LIN {X 0,Y 254.332,Z 467.701,A -85,B 0,C 180,E1 -18449.998,E2 -18449.998} C_VEL
LIN {X 0,Y 254.199,Z 468.178,A -85,B 0,C 180,E1 -18451.583,E2 -18451.583} C_VEL
LIN {X 0,Y 254.133,Z 468.22,A -85,B 0,C 180,E1 -18453.169,E2 -18453.169} C_VEL
LIN {X 0,Y 254.085,Z 467.695,A -85,B 0,C 180,E1 -18455.277,E2 -18455.277} C_VEL
LIN {X 0,Y 254.253,Z 465.99,A -85,B 0,C 180,E1 -18457.942,E2 -18457.942} C_VEL
LIN {X 0,Y 255.044,Z 462.417,A -85,B 0,C 180,E1 -18461.12,E2 -18461.12} C_VEL
LIN {X 0,Y 256.065,Z 458.576,A -85,B 0,C 180,E1 -18463.489,E2 -18463.489} C_VEL
LIN {X 0,Y 257.677,Z 453.617,A -85,B 0,C 180,E1 -18465.826,E2 -18465.826} C_VEL
LIN {X 0,Y 259.523,Z 447.396,A -85,B 0,C 180,E1 -18468.143,E2 -18468.143} C_VEL
LIN {X 0,Y 261.76,Z 439.641,A -85,B 0,C 180,E1 -18470.427,E2 -18470.427} C_VEL
LIN {X 0,Y 264.683,Z 429.976,A -85,B 0,C 180,E1 -18472.643,E2 -18472.643} C_VEL
LIN {X 0,Y 267.429,Z 419.937,A -85,B 0,C 180,E1 -18474.449,E2 -18474.449} C_VEL
LIN {X 0,Y 270.072,Z 408.613,A -85,B 0,C 180,E1 -18476.047,E2 -18476.047} C_VEL
LIN {X 0,Y 272.396,Z 397.491,A -85,B 0,C 180,E1 -18477.254,E2 -18477.254} C_VEL
LIN {X 0,Y 274.387,Z 386.142,A -85,B 0,C 180,E1 -18478.178,E2 -18478.178} C_VEL
LIN {X 0,Y 276.099,Z 372.699,A -85,B 0,C 180,E1 -18478.953,E2 -18478.953} C_VEL
LIN {X 0,Y 277.011,Z 360.119,A -85,B 0,C 180,E1 -18479.424,E2 -18479.424} C_VEL
LIN {X 0,Y 278.882,Z 309.876,A -85,B 0,C 180,E1 -18480.736,E2 -18480.736} C_VEL
LIN {X 0,Y 275.996,Z 287.607,A -85,B 0,C 180,E1 -18481.882,E2 -18481.882} C_VEL
LIN {X 0,Y 273.894,Z 274.147,A -85,B 0,C 180,E1 -18482.654,E2 -18482.654} C_VEL
LIN {X 0,Y 266.764,Z 255.183,A -85,B 0,C 180,E1 -18484.501,E2 -18484.501} C_VEL
LIN {X 0,Y 260.562,Z 245.546,A -85,B 0,C 180,E1 -18485.985,E2 -18485.985} C_VEL
LIN {X 0,Y 258.11,Z 241.688,A -85,B 0,C 180,E1 -18486.642,E2 -18486.642} C_VEL
LIN {X 0,Y 256.399,Z 238.938,A -85,B 0,C 180,E1 -18487.143,E2 -18487.143} C_VEL
LIN {X 0,Y 256.108,Z 237.583,A -85,B 0,C 180,E1 -18487.317,E2 -18487.317} C_VEL
LIN {X 0,Y 256.024,Z 237.584,A -85,B 0,C 180,E1 -18492.17,E2 -18492.17} C_VEL
LIN {X 0,Y 256.015,Z 237.588,A -85,B 0,C 180,E1 -18496.663,E2 -18496.663} C_VEL
LIN {X 0,Y 256.059,Z 237.588,A -85,B 0,C 180,E1 -18500.856,E2 -18500.856} C_VEL
LIN {X 0,Y 256.118,Z 237.562,A -85,B 0,C 180,E1 -18502.866,E2 -18502.866} C_VEL
LIN {X 0,Y 256.058,Z 237.583,A -85,B 0,C 180,E1 -18506.706,E2 -18506.706} C_VEL
LIN {X 0,Y 256.032,Z 237.558,A -85,B 0,C 180,E1 -18510.39,E2 -18510.39} C_VEL
LIN {X 0,Y 256.122,Z 237.573,A -85,B 0,C 180,E1 -18514.889,E2 -18514.889} C_VEL
LIN {X 0,Y 256.115,Z 237.547,A -85,B 0,C 180,E1 -18519.101,E2 -18519.101} C_VEL
LIN {X 0,Y 256.222,Z 237.547,A -85,B 0,C 180,E1 -18524.08,E2 -18524.08} C_VEL
LIN {X 0,Y 256.282,Z 237.553,A -85,B 0,C 180,E1 -18528.933,E2 -18528.933} C_VEL
LIN {X 0,Y 256.459,Z 237.526,A -85,B 0,C 180,E1 -18532.125,E2 -18532.125} C_VEL
LIN {X 0,Y 256.451,Z 237.522,A -85,B 0,C 180,E1 -18536.858,E2 -18536.858} C_VEL
LIN {X 0,Y 256.691,Z 237.508,A -85,B 0,C 180,E1 -18538.431,E2 -18538.431} C_VEL
LIN {X 0,Y 256.694,Z 237.476,A -85,B 0,C 180,E1 -18541.569,E2 -18541.569} C_VEL
LIN {X 0,Y 256.461,Z 237.529,A -85,B 0,C 180,E1 -18546.735,E2 -18546.735} C_VEL
LIN {X 0,Y 256.419,Z 237.512,A -85,B 0,C 180,E1 -18549.466,E2 -18549.466} C_VEL
LIN {X 0,Y 256.231,Z 237.564,A -85,B 0,C 180,E1 -18554.292,E2 -18554.292} C_VEL
LIN {X 0,Y 256.175,Z 237.545,A -85,B 0,C 180,E1 -18557.565,E2 -18557.565} C_VEL
LIN {X 0,Y 256.15,Z 237.578,A -85,B 0,C 180,E1 -18561.121,E2 -18561.121} C_VEL
LIN {X 0,Y 256.182,Z 237.56,A -85,B 0,C 180,E1 -18565.14,E2 -18565.14} C_VEL
LIN {X 0,Y 256.098,Z 237.567,A -85,B 0,C 180,E1 -18569.602,E2 -18569.602} C_VEL
LIN {X 0,Y 256.062,Z 237.579,A -85,B 0,C 180,E1 -18573.294,E2 -18573.294} C_VEL
LIN {X 0,Y 256.116,Z 237.579,A -85,B 0,C 180,E1 -18577.274,E2 -18577.274} C_VEL
LIN {X 0,Y 256.071,Z 237.583,A -85,B 0,C 180,E1 -18579.238,E2 -18579.238} C_VEL
LIN {X 0,Y 257.093,Z 240.49,A -85,B 0,C 180,E1 -18579.558,E2 -18579.558} C_VEL
LIN {X 0,Y 259.057,Z 242.91,A -85,B 0,C 180,E1 -18580.037,E2 -18580.037} C_VEL
LIN {X 0,Y 261.326,Z 246.338,A -85,B 0,C 180,E1 -18580.6,E2 -18580.6} C_VEL
LIN {X 0,Y 270.947,Z 261.865,A -85,B 0,C 180,E1 -18582.863,E2 -18582.863} C_VEL
LIN {X 0,Y 279.224,Z 277.008,A -85,B 0,C 180,E1 -18584.684,E2 -18584.684} C_VEL
LIN {X 0,Y 280.664,Z 279.841,A -85,B 0,C 180,E1 -18584.991,E2 -18584.991} C_VEL
LIN {X 0,Y 277.97,Z 342.078,A -85,B 0,C 180,E1 -18586.575,E2 -18586.575} C_VEL
LIN {X 0,Y 276.996,Z 355.523,A -85,B 0,C 180,E1 -18587.178,E2 -18587.178} C_VEL
LIN {X 0,Y 275.637,Z 367.061,A -85,B 0,C 180,E1 -18587.947,E2 -18587.947} C_VEL
LIN {X 0,Y 273.694,Z 379.563,A -85,B 0,C 180,E1 -18589.098,E2 -18589.098} C_VEL
LIN {X 0,Y 271.536,Z 390.525,A -85,B 0,C 180,E1 -18590.408,E2 -18590.408} C_VEL
LIN {X 0,Y 268.892,Z 401.605,A -85,B 0,C 180,E1 -18592.107,E2 -18592.107} C_VEL
LIN {X 0,Y 266.236,Z 411.466,A -85,B 0,C 180,E1 -18594.033,E2 -18594.033} C_VEL
LIN {X 0,Y 263.862,Z 419.47,A -85,B 0,C 180,E1 -18595.992,E2 -18595.992} C_VEL
LIN {X 0,Y 261.372,Z 427.169,A -85,B 0,C 180,E1 -18598.379,E2 -18598.379} C_VEL
LIN {X 0,Y 259.283,Z 433.28,A -85,B 0,C 180,E1 -18600.8,E2 -18600.8} C_VEL
LIN {X 0,Y 257.608,Z 438.031,A -85,B 0,C 180,E1 -18603.249,E2 -18603.249} C_VEL
LIN {X 0,Y 256.26,Z 441.573,A -85,B 0,C 180,E1 -18605.711,E2 -18605.711} C_VEL
LIN {X 0,Y 255.556,Z 443.304,A -85,B 0,C 180,E1 -18607.358,E2 -18607.358} C_VEL
LIN {X 0,Y 254.774,Z 445.019,A -85,B 0,C 180,E1 -18609.703,E2 -18609.703} C_VEL
LIN {X 0,Y 254.185,Z 445.88,A -85,B 0,C 180,E1 -18612.295,E2 -18612.295} C_VEL
LIN {X 0,Y 254.019,Z 445.872,A -85,B 0,C 180,E1 -18613.94,E2 -18613.94} C_VEL
LIN {X 0,Y 253.95,Z 445.458,A -85,B 0,C 180,E1 -18615.61,E2 -18615.61} C_VEL
LIN {X 0,Y 253.929,Z 444.63,A -85,B 0,C 180,E1 -18617.21,E2 -18617.21} C_VEL
LIN {X 0,Y 253.971,Z 443.362,A -85,B 0,C 180,E1 -18618.833,E2 -18618.833} C_VEL
LIN {X 0,Y 254.283,Z 440.661,A -85,B 0,C 180,E1 -18621.258,E2 -18621.258} C_VEL
LIN {X 0,Y 254.758,Z 436.93,A -85,B 0,C 180,E1 -18623.666,E2 -18623.666} C_VEL
LIN {X 0,Y 255.357,Z 432.082,A -85,B 0,C 180,E1 -18626.056,E2 -18626.056} C_VEL
LIN {X 0,Y 256.233,Z 425.967,A -85,B 0,C 180,E1 -18628.43,E2 -18628.43} C_VEL
LIN {X 0,Y 257.432,Z 418.31,A -85,B 0,C 180,E1 -18630.784,E2 -18630.784} C_VEL
LIN {X 0,Y 258.949,Z 408.727,A -85,B 0,C 180,E1 -18633.113,E2 -18633.113} C_VEL
LIN {X 0,Y 260.486,Z 398.784,A -85,B 0,C 180,E1 -18635.032,E2 -18635.032} C_VEL
LIN {X 0,Y 262.061,Z 387.521,A -85,B 0,C 180,E1 -18636.749,E2 -18636.749} C_VEL
LIN {X 0,Y 263.373,Z 376.65,A -85,B 0,C 180,E1 -18638.055,E2 -18638.055} C_VEL
LIN {X 0,Y 264.412,Z 364.482,A -85,B 0,C 180,E1 -18639.178,E2 -18639.178} C_VEL
LIN {X 0,Y 265.375,Z 350.98,A -85,B 0,C 180,E1 -18640.058,E2 -18640.058} C_VEL
LIN {X 0,Y 265.953,Z 338.628,A -85,B 0,C 180,E1 -18640.565,E2 -18640.565} C_VEL
LIN {X 0,Y 268.031,Z 266.062,A -85,B 0,C 180,E1 -18642.468,E2 -18642.468} C_VEL
LIN {X 0,Y 258.649,Z 243.319,A -85,B 0,C 180,E1 -18643.978,E2 -18643.978} C_VEL
LIN {X 0,Y 256.398,Z 238.283,A -85,B 0,C 180,E1 -18644.346,E2 -18644.346} C_VEL
LIN {X 0,Y 256.287,Z 237.561,A -85,B 0,C 180,E1 -18644.391,E2 -18644.391} C_VEL
LIN {X 0,Y 256.216,Z 237.569,A -85,B 0,C 180,E1 -18647.563,E2 -18647.563} C_VEL
LIN {X 0,Y 256.157,Z 237.576,A -85,B 0,C 180,E1 -18651.117,E2 -18651.117} C_VEL
LIN {X 0,Y 256.092,Z 237.584,A -85,B 0,C 180,E1 -18655.091,E2 -18655.091} C_VEL
LIN {X 0,Y 256.082,Z 237.586,A -85,B 0,C 180,E1 -18658.57,E2 -18658.57} C_VEL
LIN {X 0,Y 256.076,Z 237.584,A -85,B 0,C 180,E1 -18661.701,E2 -18661.701} C_VEL
LIN {X 0,Y 256.085,Z 237.584,A -85,B 0,C 180,E1 -18665.194,E2 -18665.194} C_VEL
LIN {X 0,Y 256.111,Z 237.578,A -85,B 0,C 180,E1 -18667.268,E2 -18667.268} C_VEL
LIN {X 0,Y 256.025,Z 237.592,A -85,B 0,C 180,E1 -18671.211,E2 -18671.211} C_VEL
LIN {X 0,Y 256.024,Z 237.593,A -85,B 0,C 180,E1 -18675.54,E2 -18675.54} C_VEL
LIN {X 0,Y 256.015,Z 237.592,A -85,B 0,C 180,E1 -18678.788,E2 -18678.788} C_VEL
LIN {X 0,Y 256.105,Z 237.573,A -85,B 0,C 180,E1 -18682.862,E2 -18682.862} C_VEL
LIN {X 0,Y 256.072,Z 237.586,A -85,B 0,C 180,E1 -18686.707,E2 -18686.707} C_VEL
LIN {X 0,Y 256.048,Z 237.582,A -85,B 0,C 180,E1 -18690.391,E2 -18690.391} C_VEL
LIN {X 0,Y 256.189,Z 237.561,A -85,B 0,C 180,E1 -18694.127,E2 -18694.127} C_VEL
LIN {X 0,Y 263.357,Z 264.994,A -85,B 0,C 180,E1 -18695.646,E2 -18695.646} C_VEL
LIN {X 0,Y 260.067,Z 344.326,A -85,B 0,C 180,E1 -18699.122,E2 -18699.122} C_VEL
LIN {X 0,Y 259.667,Z 354.656,A -85,B 0,C 180,E1 -18699.772,E2 -18699.772} C_VEL
LIN {X 0,Y 259.079,Z 358.355,A -85,B 0,C 180,E1 -18700.042,E2 -18700.042} C_VEL
LIN {X 0,Y 256.709,Z 365.442,A -85,B 0,C 180,E1 -18700.625,E2 -18700.625} C_VEL
LIN {X 0,Y 251.786,Z 377.309,A -85,B 0,C 180,E1 -18701.837,E2 -18701.837} C_VEL
LIN {X 0,Y 250.816,Z 382.417,A -85,B 0,C 180,E1 -18702.475,E2 -18702.475} C_VEL
LIN {X 0,Y 249.822,Z 394.701,A -85,B 0,C 180,E1 -18704.289,E2 -18704.289} C_VEL
LIN {X 0,Y 249.018,Z 405.731,A -85,B 0,C 180,E1 -18706.327,E2 -18706.327} C_VEL
LIN {X 0,Y 248.245,Z 415.577,A -85,B 0,C 180,E1 -18708.569,E2 -18708.569} C_VEL
LIN {X 0,Y 247.677,Z 424.27,A -85,B 0,C 180,E1 -18711.021,E2 -18711.021} C_VEL
LIN {X 0,Y 247.325,Z 431.278,A -85,B 0,C 180,E1 -18713.473,E2 -18713.473} C_VEL
LIN {X 0,Y 247.134,Z 436.857,A -85,B 0,C 180,E1 -18715.923,E2 -18715.923} C_VEL
LIN {X 0,Y 247.098,Z 441.202,A -85,B 0,C 180,E1 -18718.37,E2 -18718.37} C_VEL
LIN {X 0,Y 247.115,Z 443.466,A -85,B 0,C 180,E1 -18720,E2 -18720} C_VEL
LIN {X 0,Y 247.28,Z 445.312,A -85,B 0,C 180,E1 -18721.628,E2 -18721.628} C_VEL
LIN {X 0,Y 247.577,Z 446.731,A -85,B 0,C 180,E1 -18723.254,E2 -18723.254} C_VEL
LIN {X 0,Y 248.038,Z 447.698,A -85,B 0,C 180,E1 -18724.876,E2 -18724.876} C_VEL
LIN {X 0,Y 248.591,Z 448.265,A -85,B 0,C 180,E1 -18726.493,E2 -18726.493} C_VEL
LIN {X 0,Y 249.827,Z 448.254,A -85,B 0,C 180,E1 -18729.717,E2 -18729.717} C_VEL
LIN {X 0,Y 251.109,Z 447.597,A -85,B 0,C 180,E1 -18731.298,E2 -18731.298} C_VEL
LIN {X 0,Y 253.831,Z 445.101,A -85,B 0,C 180,E1 -18734.429,E2 -18734.429} C_VEL
LIN {X 0,Y 256.335,Z 442.134,A -85,B 0,C 180,E1 -18736.731,E2 -18736.731} C_VEL
LIN {X 0,Y 259.287,Z 438.171,A -85,B 0,C 180,E1 -18738.981,E2 -18738.981} C_VEL
LIN {X 0,Y 262.632,Z 433.126,A -85,B 0,C 180,E1 -18741.177,E2 -18741.177} C_VEL
LIN {X 0,Y 267.091,Z 425.702,A -85,B 0,C 180,E1 -18743.658,E2 -18743.658} C_VEL
LIN {X 0,Y 271.348,Z 417.742,A -85,B 0,C 180,E1 -18745.711,E2 -18745.711} C_VEL
LIN {X 0,Y 276.046,Z 408.045,A -85,B 0,C 180,E1 -18747.687,E2 -18747.687} C_VEL
LIN {X 0,Y 281.008,Z 396.101,A -85,B 0,C 180,E1 -18749.6,E2 -18749.6} C_VEL
LIN {X 0,Y 285.073,Z 384.991,A -85,B 0,C 180,E1 -18750.973,E2 -18750.973} C_VEL
LIN {X 0,Y 289.312,Z 371.238,A -85,B 0,C 180,E1 -18752.305,E2 -18752.305} C_VEL
LIN {X 0,Y 292.512,Z 358.436,A -85,B 0,C 180,E1 -18753.237,E2 -18753.237} C_VEL
LIN {X 0,Y 295.48,Z 343.206,A -85,B 0,C 180,E1 -18754.034,E2 -18754.034} C_VEL
LIN {X 0,Y 301.355,Z 311.174,A -85,B 0,C 180,E1 -18755.455,E2 -18755.455} C_VEL
LIN {X 0,Y 299.414,Z 306.995,A -85,B 0,C 180,E1 -18757.257,E2 -18757.257} C_VEL
LIN {X 0,Y 297.784,Z 304.069,A -85,B 0,C 180,E1 -18759.174,E2 -18759.174} C_VEL
LIN {X 0,Y 296.428,Z 302.2,A -85,B 0,C 180,E1 -18761.594,E2 -18761.594} C_VEL
LIN {X 0,Y 295.823,Z 302.186,A -85,B 0,C 180,E1 -18764.141,E2 -18764.141} C_VEL
LIN {X 0,Y 296.142,Z 303.62,A -85,B 0,C 180,E1 -18766.508,E2 -18766.508} C_VEL
LIN {X 0,Y 297.699,Z 309.061,A -85,B 0,C 180,E1 -18769.834,E2 -18769.834} C_VEL
LIN {X 0,Y 299.099,Z 314.072,A -85,B 0,C 180,E1 -18771.679,E2 -18771.679} C_VEL
LIN {X 0,Y 300.196,Z 318.243,A -85,B 0,C 180,E1 -18772.887,E2 -18772.887} C_VEL
LIN {X 0,Y 299.894,Z 322.243,A -85,B 0,C 180,E1 -18773.274,E2 -18773.274} C_VEL
LIN {X 0,Y 292.23,Z 364.761,A -85,B 0,C 180,E1 -18775.205,E2 -18775.205} C_VEL
LIN {X 0,Y 288.932,Z 378.053,A -85,B 0,C 180,E1 -18775.98,E2 -18775.98} C_VEL
LIN {X 0,Y 284.499,Z 392.348,A -85,B 0,C 180,E1 -18777.078,E2 -18777.078} C_VEL
LIN {X 0,Y 279.95,Z 404.975,A -85,B 0,C 180,E1 -18778.394,E2 -18778.394} C_VEL
LIN {X 0,Y 275.251,Z 416.507,A -85,B 0,C 180,E1 -18779.926,E2 -18779.926} C_VEL
LIN {X 0,Y 270.494,Z 426.944,A -85,B 0,C 180,E1 -18781.693,E2 -18781.693} C_VEL
LIN {X 0,Y 265.894,Z 436.393,A -85,B 0,C 180,E1 -18783.72,E2 -18783.72} C_VEL
LIN {X 0,Y 261.761,Z 444.205,A -85,B 0,C 180,E1 -18785.828,E2 -18785.828} C_VEL
LIN {X 0,Y 257.839,Z 451.045,A -85,B 0,C 180,E1 -18788.148,E2 -18788.148} C_VEL
LIN {X 0,Y 254.56,Z 456.733,A -85,B 0,C 180,E1 -18790.651,E2 -18790.651} C_VEL
LIN {X 0,Y 252.133,Z 460.809,A -85,B 0,C 180,E1 -18792.98,E2 -18792.98} C_VEL
LIN {X 0,Y 250.014,Z 463.933,A -85,B 0,C 180,E1 -18795.343,E2 -18795.343} C_VEL
LIN {X 0,Y 248.239,Z 466.66,A -85,B 0,C 180,E1 -18798.568,E2 -18798.568} C_VEL
LIN {X 0,Y 247.649,Z 467.451,A -85,B 0,C 180,E1 -18800.195,E2 -18800.195} C_VEL
LIN {X 0,Y 247.249,Z 467.829,A -85,B 0,C 180,E1 -18801.827,E2 -18801.827} C_VEL
LIN {X 0,Y 247.039,Z 467.373,A -85,B 0,C 180,E1 -18805.102,E2 -18805.102} C_VEL
LIN {X 0,Y 247.16,Z 465.954,A -85,B 0,C 180,E1 -18807.757,E2 -18807.757} C_VEL
LIN {X 0,Y 247.247,Z 467.319,A -85,B 0,C 180,E1 -18809.998,E2 -18809.998} C_VEL
LIN {X 0,Y 247.121,Z 467.839,A -85,B 0,C 180,E1 -18811.628,E2 -18811.628} C_VEL
LIN {X 0,Y 247.042,Z 467.918,A -85,B 0,C 180,E1 -18813.26,E2 -18813.26} C_VEL
LIN {X 0,Y 246.989,Z 467.503,A -85,B 0,C 180,E1 -18815.18,E2 -18815.18} C_VEL
LIN {X 0,Y 247.192,Z 465.788,A -85,B 0,C 180,E1 -18818.171,E2 -18818.171} C_VEL
LIN {X 0,Y 247.562,Z 464.242,A -85,B 0,C 180,E1 -18819.805,E2 -18819.805} C_VEL
LIN {X 0,Y 248.34,Z 461.149,A -85,B 0,C 180,E1 -18822.252,E2 -18822.252} C_VEL
LIN {X 0,Y 249.652,Z 457.016,A -85,B 0,C 180,E1 -18824.675,E2 -18824.675} C_VEL
LIN {X 0,Y 251.72,Z 450.712,A -85,B 0,C 180,E1 -18827.464,E2 -18827.464} C_VEL
LIN {X 0,Y 253.809,Z 443.996,A -85,B 0,C 180,E1 -18829.784,E2 -18829.784} C_VEL
LIN {X 0,Y 256.089,Z 436.905,A -85,B 0,C 180,E1 -18831.744,E2 -18831.744} C_VEL
LIN {X 0,Y 258.737,Z 428.501,A -85,B 0,C 180,E1 -18833.617,E2 -18833.617} C_VEL
LIN {X 0,Y 261.625,Z 418.133,A -85,B 0,C 180,E1 -18835.453,E2 -18835.453} C_VEL
LIN {X 0,Y 264.379,Z 406.492,A -85,B 0,C 180,E1 -18837.078,E2 -18837.078} C_VEL
LIN {X 0,Y 266.878,Z 394.749,A -85,B 0,C 180,E1 -18838.293,E2 -18838.293} C_VEL
LIN {X 0,Y 268.992,Z 382.582,A -85,B 0,C 180,E1 -18839.224,E2 -18839.224} C_VEL
LIN {X 0,Y 270.49,Z 370.041,A -85,B 0,C 180,E1 -18839.907,E2 -18839.907} C_VEL
LIN {X 0,Y 271.362,Z 355.831,A -85,B 0,C 180,E1 -18840.383,E2 -18840.383} C_VEL
LIN {X 0,Y 273.145,Z 310.97,A -85,B 0,C 180,E1 -18841.566,E2 -18841.566} C_VEL
LIN {X 0,Y 269.842,Z 284.972,A -85,B 0,C 180,E1 -18842.957,E2 -18842.957} C_VEL
LIN {X 0,Y 268.523,Z 276.891,A -85,B 0,C 180,E1 -18843.451,E2 -18843.451} C_VEL
LIN {X 0,Y 262.058,Z 259.465,A -85,B 0,C 180,E1 -18845.202,E2 -18845.202} C_VEL
LIN {X 0,Y 255.922,Z 249.902,A -85,B 0,C 180,E1 -18846.737,E2 -18846.737} C_VEL
LIN {X 0,Y 253.701,Z 246.502,A -85,B 0,C 180,E1 -18847.321,E2 -18847.321} C_VEL
LIN {X 0,Y 251.394,Z 242.907,A -85,B 0,C 180,E1 -18847.952,E2 -18847.952} C_VEL
LIN {X 0,Y 249.561,Z 240.46,A -85,B 0,C 180,E1 -18848.494,E2 -18848.494} C_VEL
LIN {X 0,Y 249.019,Z 238.452,A -85,B 0,C 180,E1 -18848.781,E2 -18848.781} C_VEL
LIN {X 0,Y 248.961,Z 238.458,A -85,B 0,C 180,E1 -18852.781,E2 -18852.781} C_VEL
LIN {X 0,Y 248.972,Z 238.455,A -85,B 0,C 180,E1 -18857.354,E2 -18857.354} C_VEL
LIN {X 0,Y 249.032,Z 238.454,A -85,B 0,C 180,E1 -18862.2,E2 -18862.2} C_VEL
LIN {X 0,Y 249.035,Z 238.445,A -85,B 0,C 180,E1 -18865.638,E2 -18865.638} C_VEL
LIN {X 0,Y 248.985,Z 238.442,A -85,B 0,C 180,E1 -18869.464,E2 -18869.464} C_VEL
LIN {X 0,Y 249.015,Z 238.453,A -85,B 0,C 180,E1 -18873.156,E2 -18873.156} C_VEL
LIN {X 0,Y 249.043,Z 238.43,A -85,B 0,C 180,E1 -18876.729,E2 -18876.729} C_VEL
LIN {X 0,Y 249.05,Z 238.443,A -85,B 0,C 180,E1 -18880.207,E2 -18880.207} C_VEL
LIN {X 0,Y 249.168,Z 238.433,A -85,B 0,C 180,E1 -18883.617,E2 -18883.617} C_VEL
LIN {X 0,Y 249.225,Z 238.428,A -85,B 0,C 180,E1 -18888.616,E2 -18888.616} C_VEL
LIN {X 0,Y 249.408,Z 238.406,A -85,B 0,C 180,E1 -18891.901,E2 -18891.901} C_VEL
LIN {X 0,Y 249.258,Z 238.397,A -85,B 0,C 180,E1 -18895.148,E2 -18895.148} C_VEL
LIN {X 0,Y 249.652,Z 238.384,A -85,B 0,C 180,E1 -18898.387,E2 -18898.387} C_VEL
LIN {X 0,Y 249.654,Z 238.352,A -85,B 0,C 180,E1 -18901.614,E2 -18901.614} C_VEL
LIN {X 0,Y 249.43,Z 238.406,A -85,B 0,C 180,E1 -18906.72,E2 -18906.72} C_VEL
LIN {X 0,Y 249.335,Z 238.391,A -85,B 0,C 180,E1 -18909.737,E2 -18909.737} C_VEL
LIN {X 0,Y 249.176,Z 238.441,A -85,B 0,C 180,E1 -18914.706,E2 -18914.706} C_VEL
LIN {X 0,Y 249.112,Z 238.427,A -85,B 0,C 180,E1 -18918.08,E2 -18918.08} C_VEL
LIN {X 0,Y 249.08,Z 238.454,A -85,B 0,C 180,E1 -18921.519,E2 -18921.519} C_VEL
LIN {X 0,Y 249.125,Z 238.444,A -85,B 0,C 180,E1 -18925.483,E2 -18925.483} C_VEL
LIN {X 0,Y 249.067,Z 238.442,A -85,B 0,C 180,E1 -18928.99,E2 -18928.99} C_VEL
LIN {X 0,Y 249.025,Z 238.465,A -85,B 0,C 180,E1 -18932.427,E2 -18932.427} C_VEL
LIN {X 0,Y 249.103,Z 238.454,A -85,B 0,C 180,E1 -18937.107,E2 -18937.107} C_VEL
LIN {X 0,Y 249.057,Z 238.556,A -85,B 0,C 180,E1 -18937.784,E2 -18937.784} C_VEL
LIN {X 0,Y 249.971,Z 241.201,A -85,B 0,C 180,E1 -18938.091,E2 -18938.091} C_VEL
LIN {X 0,Y 252.166,Z 243.937,A -85,B 0,C 180,E1 -18938.671,E2 -18938.671} C_VEL
LIN {X 0,Y 254.332,Z 247.247,A -85,B 0,C 180,E1 -18939.251,E2 -18939.251} C_VEL
LIN {X 0,Y 262.484,Z 259.993,A -85,B 0,C 180,E1 -18941.306,E2 -18941.306} C_VEL
LIN {X 0,Y 269.485,Z 271.94,A -85,B 0,C 180,E1 -18942.955,E2 -18942.955} C_VEL
LIN {X 0,Y 274.859,Z 282.268,A -85,B 0,C 180,E1 -18944.174,E2 -18944.174} C_VEL
LIN {X 0,Y 272.142,Z 342.694,A -85,B 0,C 180,E1 -18945.741,E2 -18945.741} C_VEL
LIN {X 0,Y 271.116,Z 356.115,A -85,B 0,C 180,E1 -18946.359,E2 -18946.359} C_VEL
LIN {X 0,Y 269.686,Z 367.66,A -85,B 0,C 180,E1 -18947.149,E2 -18947.149} C_VEL
LIN {X 0,Y 267.779,Z 379.415,A -85,B 0,C 180,E1 -18948.245,E2 -18948.245} C_VEL
LIN {X 0,Y 265.531,Z 390.455,A -85,B 0,C 180,E1 -18949.577,E2 -18949.577} C_VEL
LIN {X 0,Y 262.939,Z 401.008,A -85,B 0,C 180,E1 -18951.196,E2 -18951.196} C_VEL
LIN {X 0,Y 260.246,Z 410.628,A -85,B 0,C 180,E1 -18953.07,E2 -18953.07} C_VEL
LIN {X 0,Y 257.703,Z 418.826,A -85,B 0,C 180,E1 -18955.063,E2 -18955.063} C_VEL
LIN {X 0,Y 255.483,Z 425.56,A -85,B 0,C 180,E1 -18957.094,E2 -18957.094} C_VEL
LIN {X 0,Y 253.352,Z 431.504,A -85,B 0,C 180,E1 -18959.311,E2 -18959.311} C_VEL
LIN {X 0,Y 251.523,Z 436.428,A -85,B 0,C 180,E1 -18961.642,E2 -18961.642} C_VEL
LIN {X 0,Y 249.986,Z 440.404,A -85,B 0,C 180,E1 -18964.112,E2 -18964.112} C_VEL
LIN {X 0,Y 248.724,Z 443.392,A -85,B 0,C 180,E1 -18966.7,E2 -18966.7} C_VEL
LIN {X 0,Y 247.754,Z 445.352,A -85,B 0,C 180,E1 -18969.41,E2 -18969.41} C_VEL
LIN {X 0,Y 247.174,Z 446.175,A -85,B 0,C 180,E1 -18971.776,E2 -18971.776} C_VEL
LIN {X 0,Y 246.977,Z 446.22,A -85,B 0,C 180,E1 -18973.469,E2 -18973.469} C_VEL
LIN {X 0,Y 246.87,Z 445.775,A -85,B 0,C 180,E1 -18975.452,E2 -18975.452} C_VEL
LIN {X 0,Y 246.857,Z 443.911,A -85,B 0,C 180,E1 -18978.506,E2 -18978.506} C_VEL
LIN {X 0,Y 247.143,Z 441.315,A -85,B 0,C 180,E1 -18981.004,E2 -18981.004} C_VEL
LIN {X 0,Y 247.623,Z 437.693,A -85,B 0,C 180,E1 -18983.483,E2 -18983.483} C_VEL
LIN {X 0,Y 248.211,Z 432.963,A -85,B 0,C 180,E1 -18985.943,E2 -18985.943} C_VEL
LIN {X 0,Y 249.095,Z 426.976,A -85,B 0,C 180,E1 -18988.385,E2 -18988.385} C_VEL
LIN {X 0,Y 250.328,Z 419.518,A -85,B 0,C 180,E1 -18990.806,E2 -18990.806} C_VEL
LIN {X 0,Y 251.559,Z 411.884,A -85,B 0,C 180,E1 -18992.804,E2 -18992.804} C_VEL
LIN {X 0,Y 253.216,Z 401.518,A -85,B 0,C 180,E1 -18994.977,E2 -18994.977} C_VEL
LIN {X 0,Y 254.889,Z 390.698,A -85,B 0,C 180,E1 -18996.775,E2 -18996.775} C_VEL
LIN {X 0,Y 256.372,Z 379.085,A -85,B 0,C 180,E1 -18998.276,E2 -18998.276} C_VEL
LIN {X 0,Y 257.517,Z 366.588,A -85,B 0,C 180,E1 -18999.525,E2 -18999.525} C_VEL
LIN {X 0,Y 258.56,Z 353.781,A -85,B 0,C 180,E1 -19000.425,E2 -19000.425} C_VEL
LIN {X 0,Y 259.228,Z 340.348,A -85,B 0,C 180,E1 -19001.041,E2 -19001.041} C_VEL
LIN {X 0,Y 261.373,Z 267.559,A -85,B 0,C 180,E1 -19003.007,E2 -19003.007} C_VEL
LIN {X 0,Y 252.476,Z 246.187,A -85,B 0,C 180,E1 -19004.489,E2 -19004.489} C_VEL
LIN {X 0,Y 249.472,Z 239.544,A -85,B 0,C 180,E1 -19004.997,E2 -19004.997} C_VEL
LIN {X 0,Y 249.251,Z 238.437,A -85,B 0,C 180,E1 -19005.068,E2 -19005.068} C_VEL
LIN {X 0,Y 249.145,Z 238.45,A -85,B 0,C 180,E1 -19008.079,E2 -19008.079} C_VEL
LIN {X 0,Y 249.088,Z 238.457,A -85,B 0,C 180,E1 -19011.52,E2 -19011.52} C_VEL
LIN {X 0,Y 249.053,Z 238.461,A -85,B 0,C 180,E1 -19015.442,E2 -19015.442} C_VEL
LIN {X 0,Y 249.03,Z 238.464,A -85,B 0,C 180,E1 -19018.969,E2 -19018.969} C_VEL
LIN {X 0,Y 249.032,Z 238.464,A -85,B 0,C 180,E1 -19022.428,E2 -19022.428} C_VEL
LIN {X 0,Y 249.03,Z 238.459,A -85,B 0,C 180,E1 -19026.347,E2 -19026.347} C_VEL
LIN {X 0,Y 248.985,Z 238.467,A -85,B 0,C 180,E1 -19030.484,E2 -19030.484} C_VEL
LIN {X 0,Y 248.968,Z 238.467,A -85,B 0,C 180,E1 -19034.889,E2 -19034.889} C_VEL
LIN {X 0,Y 248.983,Z 238.471,A -85,B 0,C 180,E1 -19037.355,E2 -19037.355} C_VEL
LIN {X 0,Y 249.027,Z 238.452,A -85,B 0,C 180,E1 -19042.208,E2 -19042.208} C_VEL
LIN {X 0,Y 249.049,Z 238.46,A -85,B 0,C 180,E1 -19045.64,E2 -19045.64} C_VEL
LIN {X 0,Y 249,Z 238.459,A -85,B 0,C 180,E1 -19049.465,E2 -19049.465} C_VEL
LIN {X 0,Y 249.13,Z 238.44,A -85,B 0,C 180,E1 -19053.84,E2 -19053.84} C_VEL
LIN {X 0,Y 256.325,Z 266.142,A -85,B 0,C 180,E1 -19055.445,E2 -19055.445} C_VEL
LIN {X 0,Y 252.987,Z 344.975,A -85,B 0,C 180,E1 -19059.042,E2 -19059.042} C_VEL
LIN {X 0,Y 252.31,Z 359.499,A -85,B 0,C 180,E1 -19060.048,E2 -19060.048} C_VEL
LIN {X 0,Y 251.514,Z 372.185,A -85,B 0,C 180,E1 -19061.255,E2 -19061.255} C_VEL
LIN {X 0,Y 250.816,Z 382.417,A -85,B 0,C 180,E1 -19062.475,E2 -19062.475} C_VEL
LIN {X 0,Y 249.837,Z 387.422,A -85,B 0,C 180,E1 -19063.156,E2 -19063.156} C_VEL
LIN {X 0,Y 246.395,Z 395.14,A -85,B 0,C 180,E1 -19064.355,E2 -19064.355} C_VEL
LIN {X 0,Y 242.885,Z 402.444,A -85,B 0,C 180,E1 -19065.715,E2 -19065.715} C_VEL
LIN {X 0,Y 241.818,Z 406.81,A -85,B 0,C 180,E1 -19066.634,E2 -19066.634} C_VEL
LIN {X 0,Y 241.056,Z 416.98,A -85,B 0,C 180,E1 -19069.075,E2 -19069.075} C_VEL
LIN {X 0,Y 240.515,Z 425.488,A -85,B 0,C 180,E1 -19071.598,E2 -19071.598} C_VEL
LIN {X 0,Y 240.19,Z 431.628,A -85,B 0,C 180,E1 -19073.846,E2 -19073.846} C_VEL
LIN {X 0,Y 240.059,Z 437.716,A -85,B 0,C 180,E1 -19076.643,E2 -19076.643} C_VEL
LIN {X 0,Y 240.009,Z 441.943,A -85,B 0,C 180,E1 -19079.161,E2 -19079.161} C_VEL
LIN {X 0,Y 240.206,Z 445.105,A -85,B 0,C 180,E1 -19081.676,E2 -19081.676} C_VEL
LIN {X 0,Y 240.989,Z 447.81,A -85,B 0,C 180,E1 -19085.019,E2 -19085.019} C_VEL
LIN {X 0,Y 241.56,Z 448.562,A -85,B 0,C 180,E1 -19086.683,E2 -19086.683} C_VEL
LIN {X 0,Y 242.856,Z 448.833,A -85,B 0,C 180,E1 -19089.999,E2 -19089.999} C_VEL
LIN {X 0,Y 244.202,Z 448.356,A -85,B 0,C 180,E1 -19091.622,E2 -19091.622} C_VEL
LIN {X 0,Y 246.227,Z 446.97,A -85,B 0,C 180,E1 -19093.956,E2 -19093.956} C_VEL
LIN {X 0,Y 249.709,Z 443.589,A -85,B 0,C 180,E1 -19097.188,E2 -19097.188} C_VEL
LIN {X 0,Y 252.786,Z 439.951,A -85,B 0,C 180,E1 -19099.489,E2 -19099.489} C_VEL
LIN {X 0,Y 256.297,Z 435.267,A -85,B 0,C 180,E1 -19101.727,E2 -19101.727} C_VEL
LIN {X 0,Y 260.937,Z 428.305,A -85,B 0,C 180,E1 -19104.251,E2 -19104.251} C_VEL
LIN {X 0,Y 265.371,Z 420.902,A -85,B 0,C 180,E1 -19106.334,E2 -19106.334} C_VEL
LIN {X 0,Y 270.267,Z 411.853,A -85,B 0,C 180,E1 -19108.331,E2 -19108.331} C_VEL
LIN {X 0,Y 274.589,Z 402.778,A -85,B 0,C 180,E1 -19109.94,E2 -19109.94} C_VEL
LIN {X 0,Y 278.69,Z 393.113,A -85,B 0,C 180,E1 -19111.34,E2 -19111.34} C_VEL
LIN {X 0,Y 283.062,Z 381.391,A -85,B 0,C 180,E1 -19112.685,E2 -19112.685} C_VEL
LIN {X 0,Y 287.071,Z 368.438,A -85,B 0,C 180,E1 -19113.846,E2 -19113.846} C_VEL
LIN {X 0,Y 290.271,Z 355.921,A -85,B 0,C 180,E1 -19114.679,E2 -19114.679} C_VEL
LIN {X 0,Y 293.748,Z 338.33,A -85,B 0,C 180,E1 -19115.548,E2 -19115.548} C_VEL
LIN {X 0,Y 298.146,Z 315.728,A -85,B 0,C 180,E1 -19116.564,E2 -19116.564} C_VEL
LIN {X 0,Y 296.843,Z 312.974,A -85,B 0,C 180,E1 -19117.956,E2 -19117.956} C_VEL
LIN {X 0,Y 295.789,Z 310.797,A -85,B 0,C 180,E1 -19119.39,E2 -19119.39} C_VEL
LIN {X 0,Y 294.599,Z 309.061,A -85,B 0,C 180,E1 -19121.633,E2 -19121.633} C_VEL
LIN {X 0,Y 294.018,Z 309.184,A -85,B 0,C 180,E1 -19124.483,E2 -19124.483} C_VEL
LIN {X 0,Y 294.259,Z 310.576,A -85,B 0,C 180,E1 -19126.425,E2 -19126.425} C_VEL
LIN {X 0,Y 295.486,Z 315.536,A -85,B 0,C 180,E1 -19129.438,E2 -19129.438} C_VEL
LIN {X 0,Y 296.605,Z 320.223,A -85,B 0,C 180,E1 -19131.181,E2 -19131.181} C_VEL
LIN {X 0,Y 297.19,Z 322.967,A -85,B 0,C 180,E1 -19131.974,E2 -19131.974} C_VEL
LIN {X 0,Y 296.496,Z 326.882,A -85,B 0,C 180,E1 -19132.188,E2 -19132.188} C_VEL
LIN {X 0,Y 289.255,Z 364.599,A -85,B 0,C 180,E1 -19133.923,E2 -19133.923} C_VEL
LIN {X 0,Y 285.649,Z 378.062,A -85,B 0,C 180,E1 -19134.705,E2 -19134.705} C_VEL
LIN {X 0,Y 281.129,Z 391.899,A -85,B 0,C 180,E1 -19135.772,E2 -19135.772} C_VEL
LIN {X 0,Y 276.786,Z 403.223,A -85,B 0,C 180,E1 -19136.921,E2 -19136.921} C_VEL
LIN {X 0,Y 271.294,Z 415.886,A -85,B 0,C 180,E1 -19138.576,E2 -19138.576} C_VEL
LIN {X 0,Y 266.241,Z 426.256,A -85,B 0,C 180,E1 -19140.332,E2 -19140.332} C_VEL
LIN {X 0,Y 261.279,Z 435.673,A -85,B 0,C 180,E1 -19142.353,E2 -19142.353} C_VEL
LIN {X 0,Y 256.813,Z 443.481,A -85,B 0,C 180,E1 -19144.467,E2 -19144.467} C_VEL
LIN {X 0,Y 252.171,Z 450.909,A -85,B 0,C 180,E1 -19147.033,E2 -19147.033} C_VEL
LIN {X 0,Y 248.836,Z 456.041,A -85,B 0,C 180,E1 -19149.325,E2 -19149.325} C_VEL
LIN {X 0,Y 245.384,Z 461.306,A -85,B 0,C 180,E1 -19152.497,E2 -19152.497} C_VEL
LIN {X 0,Y 243.152,Z 464.143,A -85,B 0,C 180,E1 -19154.92,E2 -19154.92} C_VEL
LIN {X 0,Y 242.074,Z 465.551,A -85,B 0,C 180,E1 -19156.568,E2 -19156.568} C_VEL
LIN {X 0,Y 240.642,Z 467.159,A -85,B 0,C 180,E1 -19159.906,E2 -19159.906} C_VEL
LIN {X 0,Y 240.003,Z 467.242,A -85,B 0,C 180,E1 -19163.272,E2 -19163.272} C_VEL
LIN {X 0,Y 239.969,Z 466.699,A -85,B 0,C 180,E1 -19164.958,E2 -19164.958} C_VEL
LIN {X 0,Y 240.106,Z 465.251,A -85,B 0,C 180,E1 -19167.377,E2 -19167.377} C_VEL
LIN {X 0,Y 240.165,Z 466.937,A -85,B 0,C 180,E1 -19169.998,E2 -19169.998} C_VEL
LIN {X 0,Y 240.045,Z 467.486,A -85,B 0,C 180,E1 -19171.676,E2 -19171.676} C_VEL
LIN {X 0,Y 239.953,Z 467.616,A -85,B 0,C 180,E1 -19173.356,E2 -19173.356} C_VEL
LIN {X 0,Y 239.911,Z 467.294,A -85,B 0,C 180,E1 -19175.125,E2 -19175.125} C_VEL
LIN {X 0,Y 240.151,Z 465.574,A -85,B 0,C 180,E1 -19178.412,E2 -19178.412} C_VEL
LIN {X 0,Y 240.525,Z 464.082,A -85,B 0,C 180,E1 -19180.095,E2 -19180.095} C_VEL
LIN {X 0,Y 241.375,Z 461.051,A -85,B 0,C 180,E1 -19182.612,E2 -19182.612} C_VEL
LIN {X 0,Y 242.766,Z 456.984,A -85,B 0,C 180,E1 -19185.101,E2 -19185.101} C_VEL
LIN {X 0,Y 244.931,Z 450.752,A -85,B 0,C 180,E1 -19187.964,E2 -19187.964} C_VEL
LIN {X 0,Y 247.184,Z 443.99,A -85,B 0,C 180,E1 -19190.381,E2 -19190.381} C_VEL
LIN {X 0,Y 249.511,Z 437.112,A -85,B 0,C 180,E1 -19192.348,E2 -19192.348} C_VEL
LIN {X 0,Y 252.253,Z 428.836,A -85,B 0,C 180,E1 -19194.262,E2 -19194.262} C_VEL
LIN {X 0,Y 255.262,Z 418.649,A -85,B 0,C 180,E1 -19196.135,E2 -19196.135} C_VEL
LIN {X 0,Y 258.113,Z 407.204,A -85,B 0,C 180,E1 -19197.791,E2 -19197.791} C_VEL
LIN {X 0,Y 260.695,Z 395.854,A -85,B 0,C 180,E1 -19199.027,E2 -19199.027} C_VEL
LIN {X 0,Y 262.846,Z 384.129,A -85,B 0,C 180,E1 -19199.976,E2 -19199.976} C_VEL
LIN {X 0,Y 264.568,Z 371.212,A -85,B 0,C 180,E1 -19200.721,E2 -19200.721} C_VEL
LIN {X 0,Y 265.538,Z 357.811,A -85,B 0,C 180,E1 -19201.212,E2 -19201.212} C_VEL
LIN {X 0,Y 267.419,Z 311.486,A -85,B 0,C 180,E1 -19202.464,E2 -19202.464} C_VEL
LIN {X 0,Y 263.694,Z 282.281,A -85,B 0,C 180,E1 -19204.101,E2 -19204.101} C_VEL
LIN {X 0,Y 263.019,Z 279.243,A -85,B 0,C 180,E1 -19204.327,E2 -19204.327} C_VEL
LIN {X 0,Y 257.115,Z 263.146,A -85,B 0,C 180,E1 -19206.009,E2 -19206.009} C_VEL
LIN {X 0,Y 249.656,Z 251.604,A -85,B 0,C 180,E1 -19207.981,E2 -19207.981} C_VEL
LIN {X 0,Y 246.924,Z 247.622,A -85,B 0,C 180,E1 -19208.741,E2 -19208.741} C_VEL
LIN {X 0,Y 244.457,Z 243.906,A -85,B 0,C 180,E1 -19209.456,E2 -19209.456} C_VEL
LIN {X 0,Y 242.557,Z 241.458,A -85,B 0,C 180,E1 -19210.029,E2 -19210.029} C_VEL
LIN {X 0,Y 241.926,Z 239.343,A -85,B 0,C 180,E1 -19210.334,E2 -19210.334} C_VEL
LIN {X 0,Y 241.889,Z 239.341,A -85,B 0,C 180,E1 -19214.209,E2 -19214.209} C_VEL
LIN {X 0,Y 241.901,Z 239.331,A -85,B 0,C 180,E1 -19218.07,E2 -19218.07} C_VEL
LIN {X 0,Y 241.975,Z 239.328,A -85,B 0,C 180,E1 -19222.416,E2 -19222.416} C_VEL
LIN {X 0,Y 241.971,Z 239.337,A -85,B 0,C 180,E1 -19226.506,E2 -19226.506} C_VEL
LIN {X 0,Y 241.962,Z 239.308,A -85,B 0,C 180,E1 -19230.615,E2 -19230.615} C_VEL
LIN {X 0,Y 242.024,Z 239.33,A -85,B 0,C 180,E1 -19234.178,E2 -19234.178} C_VEL
LIN {X 0,Y 241.983,Z 239.301,A -85,B 0,C 180,E1 -19238.334,E2 -19238.334} C_VEL
LIN {X 0,Y 242.107,Z 239.317,A -85,B 0,C 180,E1 -19243.316,E2 -19243.316} C_VEL
LIN {X 0,Y 242.158,Z 239.302,A -85,B 0,C 180,E1 -19248.279,E2 -19248.279} C_VEL
LIN {X 0,Y 242.362,Z 239.287,A -85,B 0,C 180,E1 -19251.664,E2 -19251.664} C_VEL
LIN {X 0,Y 242.388,Z 239.259,A -85,B 0,C 180,E1 -19253.34,E2 -19253.34} C_VEL
LIN {X 0,Y 242.612,Z 239.26,A -85,B 0,C 180,E1 -19258.34,E2 -19258.34} C_VEL
LIN {X 0,Y 242.614,Z 239.227,A -85,B 0,C 180,E1 -19261.66,E2 -19261.66} C_VEL
LIN {X 0,Y 242.411,Z 239.283,A -85,B 0,C 180,E1 -19266.693,E2 -19266.693} C_VEL
LIN {X 0,Y 242.26,Z 239.271,A -85,B 0,C 180,E1 -19270.024,E2 -19270.024} C_VEL
LIN {X 0,Y 242.132,Z 239.314,A -85,B 0,C 180,E1 -19275.144,E2 -19275.144} C_VEL
LIN {X 0,Y 242.052,Z 239.31,A -85,B 0,C 180,E1 -19278.626,E2 -19278.626} C_VEL
LIN {X 0,Y 242.006,Z 239.327,A -85,B 0,C 180,E1 -19282.181,E2 -19282.181} C_VEL
LIN {X 0,Y 242.061,Z 239.327,A -85,B 0,C 180,E1 -19285.839,E2 -19285.839} C_VEL
LIN {X 0,Y 242.001,Z 239.322,A -85,B 0,C 180,E1 -19289.585,E2 -19289.585} C_VEL
LIN {X 0,Y 241.976,Z 239.331,A -85,B 0,C 180,E1 -19293.494,E2 -19293.494} C_VEL
LIN {X 0,Y 242.028,Z 239.509,A -85,B 0,C 180,E1 -19296.197,E2 -19296.197} C_VEL
LIN {X 0,Y 242.861,Z 241.9,A -85,B 0,C 180,E1 -19296.497,E2 -19296.497} C_VEL
LIN {X 0,Y 245.228,Z 244.787,A -85,B 0,C 180,E1 -19297.171,E2 -19297.171} C_VEL
LIN {X 0,Y 247.292,Z 248.025,A -85,B 0,C 180,E1 -19297.77,E2 -19297.77} C_VEL
LIN {X 0,Y 253.417,Z 257.185,A -85,B 0,C 180,E1 -19299.44,E2 -19299.44} C_VEL
LIN {X 0,Y 261.508,Z 270.378,A -85,B 0,C 180,E1 -19301.494,E2 -19301.494} C_VEL
LIN {X 0,Y 268.872,Z 284.129,A -85,B 0,C 180,E1 -19303.262,E2 -19303.262} C_VEL
LIN {X 0,Y 269.151,Z 284.744,A -85,B 0,C 180,E1 -19303.329,E2 -19303.329} C_VEL
LIN {X 0,Y 266.38,Z 343.4,A -85,B 0,C 180,E1 -19304.877,E2 -19304.877} C_VEL
LIN {X 0,Y 265.317,Z 356.417,A -85,B 0,C 180,E1 -19305.486,E2 -19305.486} C_VEL
LIN {X 0,Y 263.83,Z 368.057,A -85,B 0,C 180,E1 -19306.299,E2 -19306.299} C_VEL
LIN {X 0,Y 261.575,Z 381.054,A -85,B 0,C 180,E1 -19307.544,E2 -19307.544} C_VEL
LIN {X 0,Y 259.277,Z 391.843,A -85,B 0,C 180,E1 -19308.906,E2 -19308.906} C_VEL
LIN {X 0,Y 256.545,Z 402.251,A -85,B 0,C 180,E1 -19310.574,E2 -19310.574} C_VEL
LIN {X 0,Y 253.764,Z 411.622,A -85,B 0,C 180,E1 -19312.464,E2 -19312.464} C_VEL
LIN {X 0,Y 250.997,Z 420.118,A -85,B 0,C 180,E1 -19314.617,E2 -19314.617} C_VEL
LIN {X 0,Y 248.396,Z 427.499,A -85,B 0,C 180,E1 -19317.001,E2 -19317.001} C_VEL
LIN {X 0,Y 246.364,Z 432.746,A -85,B 0,C 180,E1 -19319.106,E2 -19319.106} C_VEL
LIN {X 0,Y 244.354,Z 437.749,A -85,B 0,C 180,E1 -19321.671,E2 -19321.671} C_VEL
LIN {X 0,Y 242.77,Z 441.527,A -85,B 0,C 180,E1 -19324.265,E2 -19324.265} C_VEL
LIN {X 0,Y 241.908,Z 443.444,A -85,B 0,C 180,E1 -19326.002,E2 -19326.002} C_VEL
LIN {X 0,Y 240.757,Z 445.679,A -85,B 0,C 180,E1 -19329.089,E2 -19329.089} C_VEL
LIN {X 0,Y 240.203,Z 446.432,A -85,B 0,C 180,E1 -19331.228,E2 -19331.228} C_VEL
LIN {X 0,Y 239.944,Z 446.568,A -85,B 0,C 180,E1 -19332.97,E2 -19332.97} C_VEL
LIN {X 0,Y 239.771,Z 446.088,A -85,B 0,C 180,E1 -19335.304,E2 -19335.304} C_VEL
LIN {X 0,Y 239.756,Z 444.46,A -85,B 0,C 180,E1 -19338.161,E2 -19338.161} C_VEL
LIN {X 0,Y 239.891,Z 442.887,A -85,B 0,C 180,E1 -19339.878,E2 -19339.878} C_VEL
LIN {X 0,Y 240.317,Z 439.721,A -85,B 0,C 180,E1 -19342.44,E2 -19342.44} C_VEL
LIN {X 0,Y 240.888,Z 435.489,A -85,B 0,C 180,E1 -19344.981,E2 -19344.981} C_VEL
LIN {X 0,Y 241.82,Z 429.074,A -85,B 0,C 180,E1 -19347.92,E2 -19347.92} C_VEL
LIN {X 0,Y 242.946,Z 422.012,A -85,B 0,C 180,E1 -19350.416,E2 -19350.416} C_VEL
LIN {X 0,Y 244.455,Z 413.217,A -85,B 0,C 180,E1 -19352.886,E2 -19352.886} C_VEL
LIN {X 0,Y 245.962,Z 404.184,A -85,B 0,C 180,E1 -19354.919,E2 -19354.919} C_VEL
LIN {X 0,Y 247.701,Z 393.499,A -85,B 0,C 180,E1 -19356.826,E2 -19356.826} C_VEL
LIN {X 0,Y 249.174,Z 383.058,A -85,B 0,C 180,E1 -19358.313,E2 -19358.313} C_VEL
LIN {X 0,Y 250.37,Z 371.69,A -85,B 0,C 180,E1 -19359.596,E2 -19359.596} C_VEL
LIN {X 0,Y 251.492,Z 359.348,A -85,B 0,C 180,E1 -19360.62,E2 -19360.62} C_VEL
LIN {X 0,Y 252.375,Z 346.144,A -85,B 0,C 180,E1 -19361.372,E2 -19361.372} C_VEL
LIN {X 0,Y 252.997,Z 328.878,A -85,B 0,C 180,E1 -19361.926,E2 -19361.926} C_VEL
LIN {X 0,Y 254.793,Z 269.22,A -85,B 0,C 180,E1 -19363.564,E2 -19363.564} C_VEL
LIN {X 0,Y 246.063,Z 248.305,A -85,B 0,C 180,E1 -19365.074,E2 -19365.074} C_VEL
LIN {X 0,Y 242.369,Z 240.19,A -85,B 0,C 180,E1 -19365.728,E2 -19365.728} C_VEL
LIN {X 0,Y 242.21,Z 239.315,A -85,B 0,C 180,E1 -19365.788,E2 -19365.788} C_VEL
LIN {X 0,Y 242.041,Z 239.335,A -85,B 0,C 180,E1 -19370.394,E2 -19370.394} C_VEL
LIN {X 0,Y 241.993,Z 239.341,A -85,B 0,C 180,E1 -19373.993,E2 -19373.993} C_VEL
LIN {X 0,Y 241.958,Z 239.344,A -85,B 0,C 180,E1 -19377.695,E2 -19377.695} C_VEL
LIN {X 0,Y 241.954,Z 239.341,A -85,B 0,C 180,E1 -19381.525,E2 -19381.525} C_VEL
LIN {X 0,Y 241.984,Z 239.338,A -85,B 0,C 180,E1 -19385.588,E2 -19385.588} C_VEL
LIN {X 0,Y 241.946,Z 239.348,A -85,B 0,C 180,E1 -19389.723,E2 -19389.723} C_VEL
LIN {X 0,Y 241.903,Z 239.346,A -85,B 0,C 180,E1 -19394.211,E2 -19394.211} C_VEL
LIN {X 0,Y 241.911,Z 239.348,A -85,B 0,C 180,E1 -19398.071,E2 -19398.071} C_VEL
LIN {X 0,Y 241.971,Z 239.33,A -85,B 0,C 180,E1 -19402.414,E2 -19402.414} C_VEL
LIN {X 0,Y 241.985,Z 239.34,A -85,B 0,C 180,E1 -19406.507,E2 -19406.507} C_VEL
LIN {X 0,Y 241.977,Z 239.328,A -85,B 0,C 180,E1 -19410.616,E2 -19410.616} C_VEL
LIN {X 0,Y 242.061,Z 239.337,A -85,B 0,C 180,E1 -19413.614,E2 -19413.614} C_VEL
LIN {X 0,Y 249.285,Z 266.745,A -85,B 0,C 180,E1 -19415.222,E2 -19415.222} C_VEL
LIN {X 0,Y 245.89,Z 345.36,A -85,B 0,C 180,E1 -19418.957,E2 -19418.957} C_VEL
LIN {X 0,Y 245.22,Z 359.776,A -85,B 0,C 180,E1 -19419.993,E2 -19419.993} C_VEL
LIN {X 0,Y 244.334,Z 373.326,A -85,B 0,C 180,E1 -19421.337,E2 -19421.337} C_VEL
LIN {X 0,Y 243.444,Z 385.723,A -85,B 0,C 180,E1 -19422.918,E2 -19422.918} C_VEL
LIN {X 0,Y 242.548,Z 397.939,A -85,B 0,C 180,E1 -19424.883,E2 -19424.883} C_VEL
LIN {X 0,Y 241.818,Z 406.81,A -85,B 0,C 180,E1 -19426.634,E2 -19426.634} C_VEL
LIN {X 0,Y 240.784,Z 411.023,A -85,B 0,C 180,E1 -19427.588,E2 -19427.588} C_VEL
LIN {X 0,Y 237.443,Z 417.324,A -85,B 0,C 180,E1 -19429.247,E2 -19429.247} C_VEL
LIN {X 0,Y 234.21,Z 423.164,A -85,B 0,C 180,E1 -19431.045,E2 -19431.045} C_VEL
LIN {X 0,Y 233.362,Z 426.581,A -85,B 0,C 180,E1 -19432.209,E2 -19432.209} C_VEL
LIN {X 0,Y 233.015,Z 433.222,A -85,B 0,C 180,E1 -19434.808,E2 -19434.808} C_VEL
LIN {X 0,Y 232.995,Z 438.529,A -85,B 0,C 180,E1 -19437.406,E2 -19437.406} C_VEL
LIN {X 0,Y 232.969,Z 442.65,A -85,B 0,C 180,E1 -19440,E2 -19440} C_VEL
LIN {X 0,Y 233.136,Z 444.816,A -85,B 0,C 180,E1 -19441.727,E2 -19441.727} C_VEL
LIN {X 0,Y 233.451,Z 446.557,A -85,B 0,C 180,E1 -19443.451,E2 -19443.451} C_VEL
LIN {X 0,Y 233.943,Z 447.842,A -85,B 0,C 180,E1 -19445.17,E2 -19445.17} C_VEL
LIN {X 0,Y 234.511,Z 448.736,A -85,B 0,C 180,E1 -19446.885,E2 -19446.885} C_VEL
LIN {X 0,Y 235.907,Z 449.392,A -85,B 0,C 180,E1 -19450.297,E2 -19450.297} C_VEL
LIN {X 0,Y 237.288,Z 449.085,A -85,B 0,C 180,E1 -19451.965,E2 -19451.965} C_VEL
LIN {X 0,Y 240.3,Z 447.314,A -85,B 0,C 180,E1 -19455.261,E2 -19455.261} C_VEL
LIN {X 0,Y 242.13,Z 445.851,A -85,B 0,C 180,E1 -19456.873,E2 -19456.873} C_VEL
LIN {X 0,Y 245.155,Z 442.861,A -85,B 0,C 180,E1 -19459.249,E2 -19459.249} C_VEL
LIN {X 0,Y 248.7,Z 438.872,A -85,B 0,C 180,E1 -19461.553,E2 -19461.553} C_VEL
LIN {X 0,Y 252.679,Z 433.835,A -85,B 0,C 180,E1 -19463.785,E2 -19463.785} C_VEL
LIN {X 0,Y 257.861,Z 426.445,A -85,B 0,C 180,E1 -19466.288,E2 -19466.288} C_VEL
LIN {X 0,Y 262.781,Z 418.564,A -85,B 0,C 180,E1 -19468.341,E2 -19468.341} C_VEL
LIN {X 0,Y 268.107,Z 409.012,A -85,B 0,C 180,E1 -19470.305,E2 -19470.305} C_VEL
LIN {X 0,Y 273.744,Z 397.269,A -85,B 0,C 180,E1 -19472.19,E2 -19472.19} C_VEL
LIN {X 0,Y 278.245,Z 386.564,A -85,B 0,C 180,E1 -19473.519,E2 -19473.519} C_VEL
LIN {X 0,Y 282.999,Z 373.129,A -85,B 0,C 180,E1 -19474.833,E2 -19474.833} C_VEL
LIN {X 0,Y 286.556,Z 360.834,A -85,B 0,C 180,E1 -19475.734,E2 -19475.734} C_VEL
LIN {X 0,Y 289.94,Z 346.055,A -85,B 0,C 180,E1 -19476.534,E2 -19476.534} C_VEL
LIN {X 0,Y 295.169,Z 320.529,A -85,B 0,C 180,E1 -19477.685,E2 -19477.685} C_VEL
LIN {X 0,Y 293.793,Z 317.512,A -85,B 0,C 180,E1 -19479.6,E2 -19479.6} C_VEL
LIN {X 0,Y 292.669,Z 315.881,A -85,B 0,C 180,E1 -19481.889,E2 -19481.889} C_VEL
LIN {X 0,Y 292.198,Z 316.101,A -85,B 0,C 180,E1 -19484.53,E2 -19484.53} C_VEL
LIN {X 0,Y 292.342,Z 317.271,A -85,B 0,C 180,E1 -19486.154,E2 -19486.154} C_VEL
LIN {X 0,Y 293.291,Z 321.987,A -85,B 0,C 180,E1 -19489.029,E2 -19489.029} C_VEL
LIN {X 0,Y 294.128,Z 326.159,A -85,B 0,C 180,E1 -19490.591,E2 -19490.591} C_VEL
LIN {X 0,Y 294.28,Z 327.066,A -85,B 0,C 180,E1 -19490.864,E2 -19490.864} C_VEL
LIN {X 0,Y 286.816,Z 363.581,A -85,B 0,C 180,E1 -19492.554,E2 -19492.554} C_VEL
LIN {X 0,Y 283.341,Z 376.1,A -85,B 0,C 180,E1 -19493.243,E2 -19493.243} C_VEL
LIN {X 0,Y 278.526,Z 390.229,A -85,B 0,C 180,E1 -19494.301,E2 -19494.301} C_VEL
LIN {X 0,Y 274.137,Z 401.154,A -85,B 0,C 180,E1 -19495.356,E2 -19495.356} C_VEL
LIN {X 0,Y 268.176,Z 414.22,A -85,B 0,C 180,E1 -19497.012,E2 -19497.012} C_VEL
LIN {X 0,Y 263.141,Z 424.053,A -85,B 0,C 180,E1 -19498.612,E2 -19498.612} C_VEL
LIN {X 0,Y 257.738,Z 433.657,A -85,B 0,C 180,E1 -19500.603,E2 -19500.603} C_VEL
LIN {X 0,Y 252.856,Z 441.668,A -85,B 0,C 180,E1 -19502.701,E2 -19502.701} C_VEL
LIN {X 0,Y 248.461,Z 448.336,A -85,B 0,C 180,E1 -19504.892,E2 -19504.892} C_VEL
LIN {X 0,Y 244.529,Z 453.832,A -85,B 0,C 180,E1 -19507.168,E2 -19507.168} C_VEL
LIN {X 0,Y 241.299,Z 458.25,A -85,B 0,C 180,E1 -19509.541,E2 -19509.541} C_VEL
LIN {X 0,Y 238.624,Z 461.713,A -85,B 0,C 180,E1 -19511.984,E2 -19511.984} C_VEL
LIN {X 0,Y 236.309,Z 464.293,A -85,B 0,C 180,E1 -19514.473,E2 -19514.473} C_VEL
LIN {X 0,Y 234.303,Z 466.367,A -85,B 0,C 180,E1 -19517.878,E2 -19517.878} C_VEL
LIN {X 0,Y 233.175,Z 466.934,A -85,B 0,C 180,E1 -19521.33,E2 -19521.33} C_VEL
LIN {X 0,Y 232.922,Z 465.907,A -85,B 0,C 180,E1 -19524.805,E2 -19524.805} C_VEL
LIN {X 0,Y 233.067,Z 464.541,A -85,B 0,C 180,E1 -19526.973,E2 -19526.973} C_VEL
LIN {X 0,Y 233.085,Z 466.553,A -85,B 0,C 180,E1 -19529.998,E2 -19529.998} C_VEL
LIN {X 0,Y 232.969,Z 467.129,A -85,B 0,C 180,E1 -19531.727,E2 -19531.727} C_VEL
LIN {X 0,Y 232.802,Z 467.111,A -85,B 0,C 180,E1 -19534.979,E2 -19534.979} C_VEL
LIN {X 0,Y 232.863,Z 466.393,A -85,B 0,C 180,E1 -19536.932,E2 -19536.932} C_VEL
LIN {X 0,Y 233.505,Z 463.919,A -85,B 0,C 180,E1 -19540.402,E2 -19540.402} C_VEL
LIN {X 0,Y 234.403,Z 460.942,A -85,B 0,C 180,E1 -19542.993,E2 -19542.993} C_VEL
LIN {X 0,Y 235.901,Z 456.941,A -85,B 0,C 180,E1 -19545.551,E2 -19545.551} C_VEL
LIN {X 0,Y 238.174,Z 450.794,A -85,B 0,C 180,E1 -19548.492,E2 -19548.492} C_VEL
LIN {X 0,Y 240.526,Z 444.117,A -85,B 0,C 180,E1 -19550.971,E2 -19550.971} C_VEL
LIN {X 0,Y 243.496,Z 435.854,A -85,B 0,C 180,E1 -19553.38,E2 -19553.38} C_VEL
LIN {X 0,Y 246.414,Z 427.344,A -85,B 0,C 180,E1 -19555.327,E2 -19555.327} C_VEL
LIN {X 0,Y 249.558,Z 416.882,A -85,B 0,C 180,E1 -19557.232,E2 -19557.232} C_VEL
LIN {X 0,Y 252.237,Z 406.53,A -85,B 0,C 180,E1 -19558.724,E2 -19558.724} C_VEL
LIN {X 0,Y 254.923,Z 395.045,A -85,B 0,C 180,E1 -19559.977,E2 -19559.977} C_VEL
LIN {X 0,Y 257.398,Z 381.906,A -85,B 0,C 180,E1 -19561.02,E2 -19561.02} C_VEL
LIN {X 0,Y 259.013,Z 369.32,A -85,B 0,C 180,E1 -19561.723,E2 -19561.723} C_VEL
LIN {X 0,Y 259.983,Z 354.281,A -85,B 0,C 180,E1 -19562.237,E2 -19562.237} C_VEL
LIN {X 0,Y 261.785,Z 312.508,A -85,B 0,C 180,E1 -19563.38,E2 -19563.38} C_VEL
LIN {X 0,Y 258.172,Z 283.311,A -85,B 0,C 180,E1 -19565.071,E2 -19565.071} C_VEL
LIN {X 0,Y 252.683,Z 267.751,A -85,B 0,C 180,E1 -19566.721,E2 -19566.721} C_VEL
LIN {X 0,Y 244.805,Z 255.442,A -85,B 0,C 180,E1 -19568.903,E2 -19568.903} C_VEL
LIN {X 0,Y 240.416,Z 249.051,A -85,B 0,C 180,E1 -19570.2,E2 -19570.2} C_VEL
LIN {X 0,Y 238.141,Z 245.606,A -85,B 0,C 180,E1 -19570.911,E2 -19570.911} C_VEL
LIN {X 0,Y 235.788,Z 242.93,A -85,B 0,C 180,E1 -19571.636,E2 -19571.636} C_VEL
LIN {X 0,Y 234.852,Z 240.221,A -85,B 0,C 180,E1 -19572.095,E2 -19572.095} C_VEL
LIN {X 0,Y 234.846,Z 240.225,A -85,B 0,C 180,E1 -19576.505,E2 -19576.505} C_VEL
LIN {X 0,Y 234.91,Z 240.223,A -85,B 0,C 180,E1 -19581.077,E2 -19581.077} C_VEL
LIN {X 0,Y 234.917,Z 240.198,A -85,B 0,C 180,E1 -19585.36,E2 -19585.36} C_VEL
LIN {X 0,Y 234.886,Z 240.197,A -85,B 0,C 180,E1 -19589.426,E2 -19589.426} C_VEL
LIN {X 0,Y 234.96,Z 240.211,A -85,B 0,C 180,E1 -19593.807,E2 -19593.807} C_VEL
LIN {X 0,Y 234.956,Z 240.175,A -85,B 0,C 180,E1 -19598.007,E2 -19598.007} C_VEL
LIN {X 0,Y 235.048,Z 240.198,A -85,B 0,C 180,E1 -19603.092,E2 -19603.092} C_VEL
LIN {X 0,Y 235.09,Z 240.174,A -85,B 0,C 180,E1 -19607.921,E2 -19607.921} C_VEL
LIN {X 0,Y 235.302,Z 240.17,A -85,B 0,C 180,E1 -19611.412,E2 -19611.412} C_VEL
LIN {X 0,Y 235.339,Z 240.138,A -85,B 0,C 180,E1 -19613.14,E2 -19613.14} C_VEL
LIN {X 0,Y 235.571,Z 240.137,A -85,B 0,C 180,E1 -19618.291,E2 -19618.291} C_VEL
LIN {X 0,Y 235.573,Z 240.103,A -85,B 0,C 180,E1 -19621.71,E2 -19621.71} C_VEL
LIN {X 0,Y 235.364,Z 240.16,A -85,B 0,C 180,E1 -19626.86,E2 -19626.86} C_VEL
LIN {X 0,Y 235.206,Z 240.148,A -85,B 0,C 180,E1 -19630.328,E2 -19630.328} C_VEL
LIN {X 0,Y 235.079,Z 240.186,A -85,B 0,C 180,E1 -19635.609,E2 -19635.609} C_VEL
LIN {X 0,Y 234.993,Z 240.196,A -85,B 0,C 180,E1 -19639.207,E2 -19639.207} C_VEL
LIN {X 0,Y 234.955,Z 240.197,A -85,B 0,C 180,E1 -19642.884,E2 -19642.884} C_VEL
LIN {X 0,Y 234.962,Z 240.218,A -85,B 0,C 180,E1 -19646.659,E2 -19646.659} C_VEL
LIN {X 0,Y 234.917,Z 240.211,A -85,B 0,C 180,E1 -19650.571,E2 -19650.571} C_VEL
LIN {X 0,Y 234.927,Z 240.232,A -85,B 0,C 180,E1 -19654.428,E2 -19654.428} C_VEL
LIN {X 0,Y 235.736,Z 242.771,A -85,B 0,C 180,E1 -19654.755,E2 -19654.755} C_VEL
LIN {X 0,Y 237.849,Z 245.112,A -85,B 0,C 180,E1 -19655.404,E2 -19655.404} C_VEL
LIN {X 0,Y 240.616,Z 249.16,A -85,B 0,C 180,E1 -19656.262,E2 -19656.262} C_VEL
LIN {X 0,Y 249.052,Z 261.747,A -85,B 0,C 180,E1 -19658.7,E2 -19658.7} C_VEL
LIN {X 0,Y 257.047,Z 274.96,A -85,B 0,C 180,E1 -19660.82,E2 -19660.82} C_VEL
LIN {X 0,Y 263.482,Z 287.033,A -85,B 0,C 180,E1 -19662.436,E2 -19662.436} C_VEL
LIN {X 0,Y 260.742,Z 343.044,A -85,B 0,C 180,E1 -19663.935,E2 -19663.935} C_VEL
LIN {X 0,Y 259.584,Z 356.71,A -85,B 0,C 180,E1 -19664.574,E2 -19664.574} C_VEL
LIN {X 0,Y 257.957,Z 368.932,A -85,B 0,C 180,E1 -19665.451,E2 -19665.451} C_VEL
LIN {X 0,Y 255.79,Z 380.927,A -85,B 0,C 180,E1 -19666.618,E2 -19666.618} C_VEL
LIN {X 0,Y 253.371,Z 391.808,A -85,B 0,C 180,E1 -19667.999,E2 -19667.999} C_VEL
LIN {X 0,Y 250.367,Z 402.804,A -85,B 0,C 180,E1 -19669.79,E2 -19669.79} C_VEL
LIN {X 0,Y 247.325,Z 412.619,A -85,B 0,C 180,E1 -19671.829,E2 -19671.829} C_VEL
LIN {X 0,Y 244.43,Z 420.96,A -85,B 0,C 180,E1 -19674.027,E2 -19674.027} C_VEL
LIN {X 0,Y 241.714,Z 428.241,A -85,B 0,C 180,E1 -19676.468,E2 -19676.468} C_VEL
LIN {X 0,Y 239.237,Z 434.327,A -85,B 0,C 180,E1 -19679.066,E2 -19679.066} C_VEL
LIN {X 0,Y 237.217,Z 439.056,A -85,B 0,C 180,E1 -19681.706,E2 -19681.706} C_VEL
LIN {X 0,Y 236.108,Z 441.512,A -85,B 0,C 180,E1 -19683.483,E2 -19683.483} C_VEL
LIN {X 0,Y 235.128,Z 443.482,A -85,B 0,C 180,E1 -19685.265,E2 -19685.265} C_VEL
LIN {X 0,Y 234.376,Z 445.012,A -85,B 0,C 180,E1 -19687.059,E2 -19687.059} C_VEL
LIN {X 0,Y 233.741,Z 446.052,A -85,B 0,C 180,E1 -19688.852,E2 -19688.852} C_VEL
LIN {X 0,Y 233.237,Z 446.678,A -85,B 0,C 180,E1 -19690.645,E2 -19690.645} C_VEL
LIN {X 0,Y 232.912,Z 446.899,A -85,B 0,C 180,E1 -19692.44,E2 -19692.44} C_VEL
LIN {X 0,Y 232.699,Z 446.406,A -85,B 0,C 180,E1 -19695.123,E2 -19695.123} C_VEL
LIN {X 0,Y 232.641,Z 444.974,A -85,B 0,C 180,E1 -19697.794,E2 -19697.794} C_VEL
LIN {X 0,Y 232.781,Z 443.487,A -85,B 0,C 180,E1 -19699.565,E2 -19699.565} C_VEL
LIN {X 0,Y 233.179,Z 440.429,A -85,B 0,C 180,E1 -19702.207,E2 -19702.207} C_VEL
LIN {X 0,Y 233.769,Z 436.307,A -85,B 0,C 180,E1 -19704.827,E2 -19704.827} C_VEL
LIN {X 0,Y 234.698,Z 430.019,A -85,B 0,C 180,E1 -19707.857,E2 -19707.857} C_VEL
LIN {X 0,Y 235.816,Z 423.161,A -85,B 0,C 180,E1 -19710.429,E2 -19710.429} C_VEL
LIN {X 0,Y 237.332,Z 414.536,A -85,B 0,C 180,E1 -19712.972,E2 -19712.972} C_VEL
LIN {X 0,Y 238.871,Z 405.71,A -85,B 0,C 180,E1 -19715.066,E2 -19715.066} C_VEL
LIN {X 0,Y 240.654,Z 395.279,A -85,B 0,C 180,E1 -19717.044,E2 -19717.044} C_VEL
LIN {X 0,Y 242.354,Z 383.747,A -85,B 0,C 180,E1 -19718.759,E2 -19718.759} C_VEL
LIN {X 0,Y 243.55,Z 373.403,A -85,B 0,C 180,E1 -19719.972,E2 -19719.972} C_VEL
LIN {X 0,Y 244.63,Z 362.327,A -85,B 0,C 180,E1 -19720.974,E2 -19720.974} C_VEL
LIN {X 0,Y 245.519,Z 349.42,A -85,B 0,C 180,E1 -19721.803,E2 -19721.803} C_VEL
LIN {X 0,Y 246.189,Z 335.424,A -85,B 0,C 180,E1 -19722.334,E2 -19722.334} C_VEL
LIN {X 0,Y 248.165,Z 270.796,A -85,B 0,C 180,E1 -19724.154,E2 -19724.154} C_VEL
LIN {X 0,Y 240.077,Z 251.397,A -85,B 0,C 180,E1 -19725.615,E2 -19725.615} C_VEL
LIN {X 0,Y 235.312,Z 241.114,A -85,B 0,C 180,E1 -19726.492,E2 -19726.492} C_VEL
LIN {X 0,Y 235.137,Z 240.195,A -85,B 0,C 180,E1 -19726.548,E2 -19726.548} C_VEL
LIN {X 0,Y 235.001,Z 240.212,A -85,B 0,C 180,E1 -19731.033,E2 -19731.033} C_VEL
LIN {X 0,Y 234.946,Z 240.216,A -85,B 0,C 180,E1 -19736.18,E2 -19736.18} C_VEL
LIN {X 0,Y 234.9,Z 240.218,A -85,B 0,C 180,E1 -19740.574,E2 -19740.574} C_VEL
LIN {X 0,Y 234.931,Z 240.218,A -85,B 0,C 180,E1 -19744.64,E2 -19744.64} C_VEL
LIN {X 0,Y 234.918,Z 240.221,A -85,B 0,C 180,E1 -19748.936,E2 -19748.936} C_VEL
LIN {X 0,Y 234.859,Z 240.22,A -85,B 0,C 180,E1 -19753.495,E2 -19753.495} C_VEL
LIN {X 0,Y 234.858,Z 240.227,A -85,B 0,C 180,E1 -19756.506,E2 -19756.506} C_VEL
LIN {X 0,Y 234.925,Z 240.207,A -85,B 0,C 180,E1 -19761.079,E2 -19761.079} C_VEL
LIN {X 0,Y 234.929,Z 240.22,A -85,B 0,C 180,E1 -19765.361,E2 -19765.361} C_VEL
LIN {X 0,Y 234.902,Z 240.214,A -85,B 0,C 180,E1 -19769.427,E2 -19769.427} C_VEL
LIN {X 0,Y 235.017,Z 240.198,A -85,B 0,C 180,E1 -19773.348,E2 -19773.348} C_VEL
LIN {X 0,Y 242.233,Z 268.098,A -85,B 0,C 180,E1 -19775.04,E2 -19775.04} C_VEL
LIN {X 0,Y 238.82,Z 345.465,A -85,B 0,C 180,E1 -19778.869,E2 -19778.869} C_VEL
LIN {X 0,Y 238.126,Z 359.869,A -85,B 0,C 180,E1 -19779.934,E2 -19779.934} C_VEL
LIN {X 0,Y 237.257,Z 372.967,A -85,B 0,C 180,E1 -19781.267,E2 -19781.267} C_VEL
LIN {X 0,Y 236.343,Z 385.665,A -85,B 0,C 180,E1 -19782.923,E2 -19782.923} C_VEL
LIN {X 0,Y 235.362,Z 398.606,A -85,B 0,C 180,E1 -19785.075,E2 -19785.075} C_VEL
LIN {X 0,Y 234.591,Z 408.049,A -85,B 0,C 180,E1 -19787.015,E2 -19787.015} C_VEL
LIN {X 0,Y 233.834,Z 418.298,A -85,B 0,C 180,E1 -19789.61,E2 -19789.61} C_VEL
LIN {X 0,Y 233.362,Z 426.581,A -85,B 0,C 180,E1 -19792.209,E2 -19792.209} C_VEL
LIN {X 0,Y 232.541,Z 429.824,A -85,B 0,C 180,E1 -19793.406,E2 -19793.406} C_VEL
LIN {X 0,Y 229.508,Z 434.386,A -85,B 0,C 180,E1 -19795.456,E2 -19795.456} C_VEL
LIN {X 0,Y 226.55,Z 438.359,A -85,B 0,C 180,E1 -19797.644,E2 -19797.644} C_VEL
LIN {X 0,Y 225.871,Z 440.623,A -85,B 0,C 180,E1 -19799.029,E2 -19799.029} C_VEL
LIN {X 0,Y 226.067,Z 444.431,A -85,B 0,C 180,E1 -19801.781,E2 -19801.781} C_VEL
LIN {X 0,Y 226.879,Z 447.801,A -85,B 0,C 180,E1 -19805.332,E2 -19805.332} C_VEL
LIN {X 0,Y 227.469,Z 448.883,A -85,B 0,C 180,E1 -19807.099,E2 -19807.099} C_VEL
LIN {X 0,Y 228.948,Z 449.838,A -85,B 0,C 180,E1 -19810.613,E2 -19810.613} C_VEL
LIN {X 0,Y 230.393,Z 449.72,A -85,B 0,C 180,E1 -19812.329,E2 -19812.329} C_VEL
LIN {X 0,Y 233.553,Z 448.368,A -85,B 0,C 180,E1 -19815.713,E2 -19815.713} C_VEL
LIN {X 0,Y 237.522,Z 445.394,A -85,B 0,C 180,E1 -19818.994,E2 -19818.994} C_VEL
LIN {X 0,Y 241.041,Z 442.105,A -85,B 0,C 180,E1 -19821.374,E2 -19821.374} C_VEL
LIN {X 0,Y 246.484,Z 436.165,A -85,B 0,C 180,E1 -19824.421,E2 -19824.421} C_VEL
LIN {X 0,Y 251.891,Z 429.282,A -85,B 0,C 180,E1 -19826.961,E2 -19826.961} C_VEL
LIN {X 0,Y 256.999,Z 421.991,A -85,B 0,C 180,E1 -19829.038,E2 -19829.038} C_VEL
LIN {X 0,Y 262.542,Z 413.13,A -85,B 0,C 180,E1 -19831.018,E2 -19831.018} C_VEL
LIN {X 0,Y 268.366,Z 402.363,A -85,B 0,C 180,E1 -19832.915,E2 -19832.915} C_VEL
LIN {X 0,Y 273.613,Z 391.322,A -85,B 0,C 180,E1 -19834.408,E2 -19834.408} C_VEL
LIN {X 0,Y 278.517,Z 379.21,A -85,B 0,C 180,E1 -19835.699,E2 -19835.699} C_VEL
LIN {X 0,Y 282.416,Z 367.629,A -85,B 0,C 180,E1 -19836.673,E2 -19836.673} C_VEL
LIN {X 0,Y 286.488,Z 352.816,A -85,B 0,C 180,E1 -19837.576,E2 -19837.576} C_VEL
LIN {X 0,Y 292.394,Z 325.795,A -85,B 0,C 180,E1 -19838.788,E2 -19838.788} C_VEL
LIN {X 0,Y 291.716,Z 324.159,A -85,B 0,C 180,E1 -19839.928,E2 -19839.928} C_VEL
LIN {X 0,Y 290.768,Z 322.692,A -85,B 0,C 180,E1 -19842.08,E2 -19842.08} C_VEL
LIN {X 0,Y 290.369,Z 323.007,A -85,B 0,C 180,E1 -19844.58,E2 -19844.58} C_VEL
LIN {X 0,Y 290.452,Z 323.97,A -85,B 0,C 180,E1 -19845.876,E2 -19845.876} C_VEL
LIN {X 0,Y 291.099,Z 328.25,A -85,B 0,C 180,E1 -19848.52,E2 -19848.52} C_VEL
LIN {X 0,Y 291.589,Z 331.165,A -85,B 0,C 180,E1 -19849.69,E2 -19849.69} C_VEL
LIN {X 0,Y 284.534,Z 363.504,A -85,B 0,C 180,E1 -19851.186,E2 -19851.186} C_VEL
LIN {X 0,Y 280.585,Z 376.732,A -85,B 0,C 180,E1 -19851.915,E2 -19851.915} C_VEL
LIN {X 0,Y 275.577,Z 390.499,A -85,B 0,C 180,E1 -19852.949,E2 -19852.949} C_VEL
LIN {X 0,Y 270.777,Z 401.643,A -85,B 0,C 180,E1 -19854.027,E2 -19854.027} C_VEL
LIN {X 0,Y 264.606,Z 414.293,A -85,B 0,C 180,E1 -19855.637,E2 -19855.637} C_VEL
LIN {X 0,Y 258.229,Z 425.713,A -85,B 0,C 180,E1 -19857.551,E2 -19857.551} C_VEL
LIN {X 0,Y 252.718,Z 434.717,A -85,B 0,C 180,E1 -19859.499,E2 -19859.499} C_VEL
LIN {X 0,Y 246.754,Z 443.532,A -85,B 0,C 180,E1 -19861.967,E2 -19861.967} C_VEL
LIN {X 0,Y 242.177,Z 449.742,A -85,B 0,C 180,E1 -19864.194,E2 -19864.194} C_VEL
LIN {X 0,Y 238.091,Z 454.853,A -85,B 0,C 180,E1 -19866.514,E2 -19866.514} C_VEL
LIN {X 0,Y 234.712,Z 458.944,A -85,B 0,C 180,E1 -19868.94,E2 -19868.94} C_VEL
LIN {X 0,Y 231.016,Z 462.969,A -85,B 0,C 180,E1 -19872.287,E2 -19872.287} C_VEL
LIN {X 0,Y 228.229,Z 465.473,A -85,B 0,C 180,E1 -19875.737,E2 -19875.737} C_VEL
LIN {X 0,Y 226.643,Z 466.436,A -85,B 0,C 180,E1 -19879.275,E2 -19879.275} C_VEL
LIN {X 0,Y 225.92,Z 465.913,A -85,B 0,C 180,E1 -19882.85,E2 -19882.85} C_VEL
LIN {X 0,Y 225.902,Z 465.09,A -85,B 0,C 180,E1 -19884.643,E2 -19884.643} C_VEL
LIN {X 0,Y 225.998,Z 463.796,A -85,B 0,C 180,E1 -19886.544,E2 -19886.544} C_VEL
LIN {X 0,Y 225.94,Z 465.155,A -85,B 0,C 180,E1 -19888.216,E2 -19888.216} C_VEL
LIN {X 0,Y 226.007,Z 466.169,A -85,B 0,C 180,E1 -19889.998,E2 -19889.998} C_VEL
LIN {X 0,Y 225.893,Z 466.773,A -85,B 0,C 180,E1 -19891.781,E2 -19891.781} C_VEL
LIN {X 0,Y 225.715,Z 466.86,A -85,B 0,C 180,E1 -19894.882,E2 -19894.882} C_VEL
LIN {X 0,Y 225.796,Z 466.147,A -85,B 0,C 180,E1 -19897.15,E2 -19897.15} C_VEL
LIN {X 0,Y 226.503,Z 463.743,A -85,B 0,C 180,E1 -19900.727,E2 -19900.727} C_VEL
LIN {X 0,Y 227.455,Z 460.821,A -85,B 0,C 180,E1 -19903.397,E2 -19903.397} C_VEL
LIN {X 0,Y 229.057,Z 456.888,A -85,B 0,C 180,E1 -19906.028,E2 -19906.028} C_VEL
LIN {X 0,Y 231.055,Z 451.829,A -85,B 0,C 180,E1 -19908.623,E2 -19908.623} C_VEL
LIN {X 0,Y 233.43,Z 445.475,A -85,B 0,C 180,E1 -19911.177,E2 -19911.177} C_VEL
LIN {X 0,Y 236.457,Z 437.56,A -85,B 0,C 180,E1 -19913.654,E2 -19913.654} C_VEL
LIN {X 0,Y 240.04,Z 427.733,A -85,B 0,C 180,E1 -19916.049,E2 -19916.049} C_VEL
LIN {X 0,Y 243.299,Z 417.423,A -85,B 0,C 180,E1 -19917.993,E2 -19917.993} C_VEL
LIN {X 0,Y 246.481,Z 405.848,A -85,B 0,C 180,E1 -19919.695,E2 -19919.695} C_VEL
LIN {X 0,Y 249.249,Z 394.231,A -85,B 0,C 180,E1 -19920.968,E2 -19920.968} C_VEL
LIN {X 0,Y 251.806,Z 380.955,A -85,B 0,C 180,E1 -19922.023,E2 -19922.023} C_VEL
LIN {X 0,Y 253.413,Z 368.328,A -85,B 0,C 180,E1 -19922.724,E2 -19922.724} C_VEL
LIN {X 0,Y 254.441,Z 352.763,A -85,B 0,C 180,E1 -19923.248,E2 -19923.248} C_VEL
LIN {X 0,Y 256.252,Z 313.661,A -85,B 0,C 180,E1 -19924.329,E2 -19924.329} C_VEL
LIN {X 0,Y 252.903,Z 285.772,A -85,B 0,C 180,E1 -19925.998,E2 -19925.998} C_VEL
LIN {X 0,Y 247.939,Z 271.72,A -85,B 0,C 180,E1 -19927.559,E2 -19927.559} C_VEL
LIN {X 0,Y 239.767,Z 258.786,A -85,B 0,C 180,E1 -19929.946,E2 -19929.946} C_VEL
LIN {X 0,Y 236.064,Z 253.605,A -85,B 0,C 180,E1 -19931.091,E2 -19931.091} C_VEL
LIN {X 0,Y 233.903,Z 250.485,A -85,B 0,C 180,E1 -19931.795,E2 -19931.795} C_VEL
LIN {X 0,Y 231.613,Z 247.321,A -85,B 0,C 180,E1 -19932.56,E2 -19932.56} C_VEL
LIN {X 0,Y 230.991,Z 246.16,A -85,B 0,C 180,E1 -19932.787,E2 -19932.787} C_VEL
LIN {X 0,Y 228.891,Z 244.07,A -85,B 0,C 180,E1 -19933.481,E2 -19933.481} C_VEL
LIN {X 0,Y 227.844,Z 241.365,A -85,B 0,C 180,E1 -19933.923,E2 -19933.923} C_VEL
LIN {X 0,Y 227.833,Z 241.09,A -85,B 0,C 180,E1 -19934.098,E2 -19934.098} C_VEL
LIN {X 0,Y 227.78,Z 241.091,A -85,B 0,C 180,E1 -19937.771,E2 -19937.771} C_VEL
LIN {X 0,Y 227.832,Z 241.097,A -85,B 0,C 180,E1 -19941.907,E2 -19941.907} C_VEL
LIN {X 0,Y 227.871,Z 241.09,A -85,B 0,C 180,E1 -19946.377,E2 -19946.377} C_VEL
LIN {X 0,Y 227.863,Z 241.063,A -85,B 0,C 180,E1 -19950.43,E2 -19950.43} C_VEL
LIN {X 0,Y 227.893,Z 241.091,A -85,B 0,C 180,E1 -19954.422,E2 -19954.422} C_VEL
LIN {X 0,Y 227.917,Z 241.051,A -85,B 0,C 180,E1 -19958.283,E2 -19958.283} C_VEL
LIN {X 0,Y 228.012,Z 241.06,A -85,B 0,C 180,E1 -19963.895,E2 -19963.895} C_VEL
LIN {X 0,Y 228.134,Z 241.063,A -85,B 0,C 180,E1 -19969.349,E2 -19969.349} C_VEL
LIN {X 0,Y 228.292,Z 241.018,A -85,B 0,C 180,E1 -19972.927,E2 -19972.927} C_VEL
LIN {X 0,Y 228.53,Z 241.013,A -85,B 0,C 180,E1 -19978.238,E2 -19978.238} C_VEL
LIN {X 0,Y 228.531,Z 240.979,A -85,B 0,C 180,E1 -19981.763,E2 -19981.763} C_VEL
LIN {X 0,Y 228.315,Z 241.038,A -85,B 0,C 180,E1 -19987.073,E2 -19987.073} C_VEL
LIN {X 0,Y 228.137,Z 241.028,A -85,B 0,C 180,E1 -19990.652,E2 -19990.652} C_VEL
LIN {X 0,Y 228.041,Z 241.075,A -85,B 0,C 180,E1 -19994.274,E2 -19994.274} C_VEL
LIN {X 0,Y 227.984,Z 241.056,A -85,B 0,C 180,E1 -19997.955,E2 -19997.955} C_VEL
LIN {X 0,Y 227.924,Z 241.078,A -85,B 0,C 180,E1 -20002.33,E2 -20002.33} C_VEL
LIN {X 0,Y 227.936,Z 241.093,A -85,B 0,C 180,E1 -20006.604,E2 -20006.604} C_VEL
LIN {X 0,Y 227.891,Z 241.083,A -85,B 0,C 180,E1 -20010.293,E2 -20010.293} C_VEL
LIN {X 0,Y 227.921,Z 241.092,A -85,B 0,C 180,E1 -20012.462,E2 -20012.462} C_VEL
LIN {X 0,Y 228.838,Z 243.811,A -85,B 0,C 180,E1 -20012.903,E2 -20012.903} C_VEL
LIN {X 0,Y 230.84,Z 245.998,A -85,B 0,C 180,E1 -20013.575,E2 -20013.575} C_VEL
LIN {X 0,Y 233.643,Z 250.105,A -85,B 0,C 180,E1 -20014.53,E2 -20014.53} C_VEL
LIN {X 0,Y 234.996,Z 251.844,A -85,B 0,C 180,E1 -20014.965,E2 -20014.965} C_VEL
LIN {X 0,Y 240.614,Z 260.007,A -85,B 0,C 180,E1 -20016.718,E2 -20016.718} C_VEL
LIN {X 0,Y 248.068,Z 271.811,A -85,B 0,C 180,E1 -20018.882,E2 -20018.882} C_VEL
LIN {X 0,Y 255.45,Z 284.816,A -85,B 0,C 180,E1 -20020.873,E2 -20020.873} C_VEL
LIN {X 0,Y 257.878,Z 289.478,A -85,B 0,C 180,E1 -20021.503,E2 -20021.503} C_VEL
LIN {X 0,Y 255.096,Z 344.112,A -85,B 0,C 180,E1 -20022.998,E2 -20022.998} C_VEL
LIN {X 0,Y 253.936,Z 357.122,A -85,B 0,C 180,E1 -20023.626,E2 -20023.626} C_VEL
LIN {X 0,Y 252.24,Z 369.21,A -85,B 0,C 180,E1 -20024.504,E2 -20024.504} C_VEL
LIN {X 0,Y 250.06,Z 380.83,A -85,B 0,C 180,E1 -20025.647,E2 -20025.647} C_VEL
LIN {X 0,Y 247.538,Z 391.785,A -85,B 0,C 180,E1 -20027.05,E2 -20027.05} C_VEL
LIN {X 0,Y 244.757,Z 401.779,A -85,B 0,C 180,E1 -20028.67,E2 -20028.67} C_VEL
LIN {X 0,Y 241.499,Z 411.805,A -85,B 0,C 180,E1 -20030.734,E2 -20030.734} C_VEL
LIN {X 0,Y 238.24,Z 420.939,A -85,B 0,C 180,E1 -20033.14,E2 -20033.14} C_VEL
LIN {X 0,Y 235.514,Z 427.849,A -85,B 0,C 180,E1 -20035.463,E2 -20035.463} C_VEL
LIN {X 0,Y 232.79,Z 434.27,A -85,B 0,C 180,E1 -20038.219,E2 -20038.219} C_VEL
LIN {X 0,Y 230.674,Z 438.926,A -85,B 0,C 180,E1 -20040.828,E2 -20040.828} C_VEL
LIN {X 0,Y 228.934,Z 442.565,A -85,B 0,C 180,E1 -20043.57,E2 -20043.57} C_VEL
LIN {X 0,Y 227.542,Z 445.11,A -85,B 0,C 180,E1 -20046.329,E2 -20046.329} C_VEL
LIN {X 0,Y 226.754,Z 446.348,A -85,B 0,C 180,E1 -20048.408,E2 -20048.408} C_VEL
LIN {X 0,Y 225.906,Z 447.198,A -85,B 0,C 180,E1 -20051.876,E2 -20051.876} C_VEL
LIN {X 0,Y 225.621,Z 446.72,A -85,B 0,C 180,E1 -20054.939,E2 -20054.939} C_VEL
LIN {X 0,Y 225.547,Z 445.469,A -85,B 0,C 180,E1 -20057.404,E2 -20057.404} C_VEL
LIN {X 0,Y 225.64,Z 444.073,A -85,B 0,C 180,E1 -20059.231,E2 -20059.231} C_VEL
LIN {X 0,Y 226.04,Z 441.118,A -85,B 0,C 180,E1 -20061.959,E2 -20061.959} C_VEL
LIN {X 0,Y 226.621,Z 437.114,A -85,B 0,C 180,E1 -20064.664,E2 -20064.664} C_VEL
LIN {X 0,Y 227.566,Z 430.947,A -85,B 0,C 180,E1 -20067.79,E2 -20067.79} C_VEL
LIN {X 0,Y 228.664,Z 424.237,A -85,B 0,C 180,E1 -20070.442,E2 -20070.442} C_VEL
LIN {X 0,Y 229.925,Z 417.371,A -85,B 0,C 180,E1 -20072.63,E2 -20072.63} C_VEL
LIN {X 0,Y 231.448,Z 409.095,A -85,B 0,C 180,E1 -20074.792,E2 -20074.792} C_VEL
LIN {X 0,Y 233.299,Z 398.87,A -85,B 0,C 180,E1 -20076.923,E2 -20076.923} C_VEL
LIN {X 0,Y 235.133,Z 387.419,A -85,B 0,C 180,E1 -20078.813,E2 -20078.813} C_VEL
LIN {X 0,Y 236.627,Z 376.021,A -85,B 0,C 180,E1 -20080.267,E2 -20080.267} C_VEL
LIN {X 0,Y 237.763,Z 364.426,A -85,B 0,C 180,E1 -20081.403,E2 -20081.403} C_VEL
LIN {X 0,Y 238.836,Z 351.131,A -85,B 0,C 180,E1 -20082.325,E2 -20082.325} C_VEL
LIN {X 0,Y 239.495,Z 338.121,A -85,B 0,C 180,E1 -20082.872,E2 -20082.872} C_VEL
LIN {X 0,Y 241.662,Z 272.635,A -85,B 0,C 180,E1 -20084.757,E2 -20084.757} C_VEL
LIN {X 0,Y 234.043,Z 254.319,A -85,B 0,C 180,E1 -20086.196,E2 -20086.196} C_VEL
LIN {X 0,Y 228.209,Z 241.915,A -85,B 0,C 180,E1 -20087.312,E2 -20087.312} C_VEL
LIN {X 0,Y 228.042,Z 241.079,A -85,B 0,C 180,E1 -20087.445,E2 -20087.445} C_VEL
LIN {X 0,Y 227.916,Z 241.093,A -85,B 0,C 180,E1 -20092.318,E2 -20092.318} C_VEL
LIN {X 0,Y 227.907,Z 241.092,A -85,B 0,C 180,E1 -20096.583,E2 -20096.583} C_VEL
LIN {X 0,Y 227.875,Z 241.094,A -85,B 0,C 180,E1 -20100.28,E2 -20100.28} C_VEL
LIN {X 0,Y 227.882,Z 241.101,A -85,B 0,C 180,E1 -20103.722,E2 -20103.722} C_VEL
LIN {X 0,Y 227.846,Z 241.103,A -85,B 0,C 180,E1 -20108.093,E2 -20108.093} C_VEL
LIN {X 0,Y 227.792,Z 241.098,A -85,B 0,C 180,E1 -20112.749,E2 -20112.749} C_VEL
LIN {X 0,Y 227.79,Z 241.111,A -85,B 0,C 180,E1 -20117.252,E2 -20117.252} C_VEL
LIN {X 0,Y 227.844,Z 241.088,A -85,B 0,C 180,E1 -20121.908,E2 -20121.908} C_VEL
LIN {X 0,Y 227.885,Z 241.096,A -85,B 0,C 180,E1 -20126.378,E2 -20126.378} C_VEL
LIN {X 0,Y 227.88,Z 241.084,A -85,B 0,C 180,E1 -20130.432,E2 -20130.432} C_VEL
LIN {X 0,Y 227.952,Z 241.073,A -85,B 0,C 180,E1 -20133.101,E2 -20133.101} C_VEL
LIN {X 0,Y 235.181,Z 268.677,A -85,B 0,C 180,E1 -20134.83,E2 -20134.83} C_VEL
LIN {X 0,Y 231.759,Z 345.244,A -85,B 0,C 180,E1 -20138.776,E2 -20138.776} C_VEL
LIN {X 0,Y 231.056,Z 359.68,A -85,B 0,C 180,E1 -20139.873,E2 -20139.873} C_VEL
LIN {X 0,Y 230.237,Z 372.003,A -85,B 0,C 180,E1 -20141.139,E2 -20141.139} C_VEL
LIN {X 0,Y 229.304,Z 384.883,A -85,B 0,C 180,E1 -20142.842,E2 -20142.842} C_VEL
LIN {X 0,Y 228.426,Z 396.828,A -85,B 0,C 180,E1 -20144.839,E2 -20144.839} C_VEL
LIN {X 0,Y 227.52,Z 407.585,A -85,B 0,C 180,E1 -20147.058,E2 -20147.058} C_VEL
LIN {X 0,Y 226.9,Z 416.439,A -85,B 0,C 180,E1 -20149.289,E2 -20149.289} C_VEL
LIN {X 0,Y 226.306,Z 425.91,A -85,B 0,C 180,E1 -20152.249,E2 -20152.249} C_VEL
LIN {X 0,Y 225.977,Z 432.105,A -85,B 0,C 180,E1 -20154.646,E2 -20154.646} C_VEL
LIN {X 0,Y 225.931,Z 437.727,A -85,B 0,C 180,E1 -20157.325,E2 -20157.325} C_VEL
LIN {X 0,Y 225.871,Z 440.623,A -85,B 0,C 180,E1 -20159.029,E2 -20159.029} C_VEL
LIN {X 0,Y 225.249,Z 442.703,A -85,B 0,C 180,E1 -20160.424,E2 -20160.424} C_VEL
LIN {X 0,Y 222.676,Z 445.395,A -85,B 0,C 180,E1 -20162.775,E2 -20162.775} C_VEL
LIN {X 0,Y 220.695,Z 447.073,A -85,B 0,C 180,E1 -20164.728,E2 -20164.728} C_VEL
LIN {X 0,Y 220.118,Z 448.211,A -85,B 0,C 180,E1 -20166.241,E2 -20166.241} C_VEL
LIN {X 0,Y 220.213,Z 448.499,A -85,B 0,C 180,E1 -20166.748,E2 -20166.748} C_VEL
LIN {X 0,Y 221.072,Z 449.75,A -85,B 0,C 180,E1 -20169.146,E2 -20169.146} C_VEL
LIN {X 0,Y 222.004,Z 450.239,A -85,B 0,C 180,E1 -20170.949,E2 -20170.949} C_VEL
LIN {X 0,Y 223.487,Z 450.321,A -85,B 0,C 180,E1 -20172.716,E2 -20172.716} C_VEL
LIN {X 0,Y 226.8,Z 449.306,A -85,B 0,C 180,E1 -20176.194,E2 -20176.194} C_VEL
LIN {X 0,Y 230.967,Z 446.794,A -85,B 0,C 180,E1 -20179.555,E2 -20179.555} C_VEL
LIN {X 0,Y 234.639,Z 443.836,A -85,B 0,C 180,E1 -20181.987,E2 -20181.987} C_VEL
LIN {X 0,Y 238.84,Z 439.909,A -85,B 0,C 180,E1 -20184.328,E2 -20184.328} C_VEL
LIN {X 0,Y 243.464,Z 434.96,A -85,B 0,C 180,E1 -20186.579,E2 -20186.579} C_VEL
LIN {X 0,Y 249.418,Z 427.737,A -85,B 0,C 180,E1 -20189.082,E2 -20189.082} C_VEL
LIN {X 0,Y 255.136,Z 419.873,A -85,B 0,C 180,E1 -20191.143,E2 -20191.143} C_VEL
LIN {X 0,Y 261.217,Z 410.382,A -85,B 0,C 180,E1 -20193.112,E2 -20193.112} C_VEL
LIN {X 0,Y 267.05,Z 399.888,A -85,B 0,C 180,E1 -20194.803,E2 -20194.803} C_VEL
LIN {X 0,Y 272.923,Z 387.698,A -85,B 0,C 180,E1 -20196.318,E2 -20196.318} C_VEL
LIN {X 0,Y 278.124,Z 374.756,A -85,B 0,C 180,E1 -20197.562,E2 -20197.562} C_VEL
LIN {X 0,Y 282.383,Z 361.866,A -85,B 0,C 180,E1 -20198.477,E2 -20198.477} C_VEL
LIN {X 0,Y 286.216,Z 346.891,A -85,B 0,C 180,E1 -20199.264,E2 -20199.264} C_VEL
LIN {X 0,Y 289.862,Z 331.032,A -85,B 0,C 180,E1 -20199.946,E2 -20199.946} C_VEL
LIN {X 0,Y 288.947,Z 329.549,A -85,B 0,C 180,E1 -20202.068,E2 -20202.068} C_VEL
LIN {X 0,Y 288.541,Z 329.764,A -85,B 0,C 180,E1 -20204.327,E2 -20204.327} C_VEL
LIN {X 0,Y 288.563,Z 330.652,A -85,B 0,C 180,E1 -20205.569,E2 -20205.569} C_VEL
LIN {X 0,Y 288.981,Z 334.674,A -85,B 0,C 180,E1 -20208.089,E2 -20208.089} C_VEL
LIN {X 0,Y 289.082,Z 335.707,A -85,B 0,C 180,E1 -20208.503,E2 -20208.503} C_VEL
LIN {X 0,Y 282.48,Z 364.001,A -85,B 0,C 180,E1 -20209.809,E2 -20209.809} C_VEL
LIN {X 0,Y 278.043,Z 377.742,A -85,B 0,C 180,E1 -20210.573,E2 -20210.573} C_VEL
LIN {X 0,Y 272.83,Z 391.096,A -85,B 0,C 180,E1 -20211.576,E2 -20211.576} C_VEL
LIN {X 0,Y 267.19,Z 403.264,A -85,B 0,C 180,E1 -20212.771,E2 -20212.771} C_VEL
LIN {X 0,Y 260.453,Z 415.893,A -85,B 0,C 180,E1 -20214.429,E2 -20214.429} C_VEL
LIN {X 0,Y 253.73,Z 427.01,A -85,B 0,C 180,E1 -20216.358,E2 -20216.358} C_VEL
LIN {X 0,Y 246.83,Z 437.147,A -85,B 0,C 180,E1 -20218.69,E2 -20218.69} C_VEL
LIN {X 0,Y 240.668,Z 445.36,A -85,B 0,C 180,E1 -20221.193,E2 -20221.193} C_VEL
LIN {X 0,Y 235.912,Z 451.128,A -85,B 0,C 180,E1 -20223.456,E2 -20223.456} C_VEL
LIN {X 0,Y 231.684,Z 455.857,A -85,B 0,C 180,E1 -20225.824,E2 -20225.824} C_VEL
LIN {X 0,Y 228.133,Z 459.601,A -85,B 0,C 180,E1 -20228.302,E2 -20228.302} C_VEL
LIN {X 0,Y 224.277,Z 463.203,A -85,B 0,C 180,E1 -20231.736,E2 -20231.736} C_VEL
LIN {X 0,Y 221.331,Z 465.316,A -85,B 0,C 180,E1 -20235.282,E2 -20235.282} C_VEL
LIN {X 0,Y 219.652,Z 465.989,A -85,B 0,C 180,E1 -20238.93,E2 -20238.93} C_VEL
LIN {X 0,Y 218.908,Z 465.136,A -85,B 0,C 180,E1 -20242.62,E2 -20242.62} C_VEL
LIN {X 0,Y 218.96,Z 462.983,A -85,B 0,C 180,E1 -20246.077,E2 -20246.077} C_VEL
LIN {X 0,Y 218.875,Z 464.731,A -85,B 0,C 180,E1 -20248.158,E2 -20248.158} C_VEL
LIN {X 0,Y 218.931,Z 465.784,A -85,B 0,C 180,E1 -20249.998,E2 -20249.998} C_VEL
LIN {X 0,Y 218.818,Z 466.416,A -85,B 0,C 180,E1 -20251.839,E2 -20251.839} C_VEL
LIN {X 0,Y 218.648,Z 466.495,A -85,B 0,C 180,E1 -20255.532,E2 -20255.532} C_VEL
LIN {X 0,Y 219.006,Z 464.925,A -85,B 0,C 180,E1 -20259.231,E2 -20259.231} C_VEL
LIN {X 0,Y 219.497,Z 463.559,A -85,B 0,C 180,E1 -20261.074,E2 -20261.074} C_VEL
LIN {X 0,Y 220.528,Z 460.699,A -85,B 0,C 180,E1 -20263.826,E2 -20263.826} C_VEL
LIN {X 0,Y 222.234,Z 456.831,A -85,B 0,C 180,E1 -20266.534,E2 -20266.534} C_VEL
LIN {X 0,Y 224.33,Z 451.844,A -85,B 0,C 180,E1 -20269.203,E2 -20269.203} C_VEL
LIN {X 0,Y 226.827,Z 445.595,A -85,B 0,C 180,E1 -20271.825,E2 -20271.825} C_VEL
LIN {X 0,Y 229.965,Z 437.79,A -85,B 0,C 180,E1 -20274.364,E2 -20274.364} C_VEL
LIN {X 0,Y 233.706,Z 428.088,A -85,B 0,C 180,E1 -20276.811,E2 -20276.811} C_VEL
LIN {X 0,Y 237.089,Z 417.981,A -85,B 0,C 180,E1 -20278.794,E2 -20278.794} C_VEL
LIN {X 0,Y 240.375,Z 406.602,A -85,B 0,C 180,E1 -20280.529,E2 -20280.529} C_VEL
LIN {X 0,Y 243.244,Z 395.385,A -85,B 0,C 180,E1 -20281.82,E2 -20281.82} C_VEL
LIN {X 0,Y 245.881,Z 382.576,A -85,B 0,C 180,E1 -20282.891,E2 -20282.891} C_VEL
LIN {X 0,Y 247.708,Z 369.838,A -85,B 0,C 180,E1 -20283.65,E2 -20283.65} C_VEL
LIN {X 0,Y 248.782,Z 355.808,A -85,B 0,C 180,E1 -20284.176,E2 -20284.176} C_VEL
LIN {X 0,Y 250.723,Z 314.486,A -85,B 0,C 180,E1 -20285.348,E2 -20285.348} C_VEL
LIN {X 0,Y 247.679,Z 288.206,A -85,B 0,C 180,E1 -20286.969,E2 -20286.969} C_VEL
LIN {X 0,Y 243.446,Z 276.045,A -85,B 0,C 180,E1 -20288.375,E2 -20288.375} C_VEL
LIN {X 0,Y 235.81,Z 263.809,A -85,B 0,C 180,E1 -20290.709,E2 -20290.709} C_VEL
LIN {X 0,Y 230.137,Z 255.702,A -85,B 0,C 180,E1 -20292.581,E2 -20292.581} C_VEL
LIN {X 0,Y 227.063,Z 251.458,A -85,B 0,C 180,E1 -20293.658,E2 -20293.658} C_VEL
LIN {X 0,Y 224.76,Z 248.33,A -85,B 0,C 180,E1 -20294.498,E2 -20294.498} C_VEL
LIN {X 0,Y 223.931,Z 247.051,A -85,B 0,C 180,E1 -20294.816,E2 -20294.816} C_VEL
LIN {X 0,Y 221.741,Z 244.846,A -85,B 0,C 180,E1 -20295.618,E2 -20295.618} C_VEL
LIN {X 0,Y 220.813,Z 242.573,A -85,B 0,C 180,E1 -20296.036,E2 -20296.036} C_VEL
LIN {X 0,Y 220.712,Z 241.99,A -85,B 0,C 180,E1 -20296.17,E2 -20296.17} C_VEL
LIN {X 0,Y 220.774,Z 241.979,A -85,B 0,C 180,E1 -20300.456,E2 -20300.456} C_VEL
LIN {X 0,Y 220.818,Z 241.956,A -85,B 0,C 180,E1 -20302.792,E2 -20302.792} C_VEL
LIN {X 0,Y 220.803,Z 241.977,A -85,B 0,C 180,E1 -20307.242,E2 -20307.242} C_VEL
LIN {X 0,Y 220.791,Z 241.945,A -85,B 0,C 180,E1 -20311.48,E2 -20311.48} C_VEL
LIN {X 0,Y 220.836,Z 241.957,A -85,B 0,C 180,E1 -20315.562,E2 -20315.562} C_VEL
LIN {X 0,Y 220.845,Z 241.94,A -85,B 0,C 180,E1 -20319.51,E2 -20319.51} C_VEL
LIN {X 0,Y 220.969,Z 241.946,A -85,B 0,C 180,E1 -20323.367,E2 -20323.367} C_VEL
LIN {X 0,Y 221.054,Z 241.94,A -85,B 0,C 180,E1 -20329.003,E2 -20329.003} C_VEL
LIN {X 0,Y 221.23,Z 241.899,A -85,B 0,C 180,E1 -20332.7,E2 -20332.7} C_VEL
LIN {X 0,Y 221.463,Z 241.893,A -85,B 0,C 180,E1 -20338.182,E2 -20338.182} C_VEL
LIN {X 0,Y 221.465,Z 241.857,A -85,B 0,C 180,E1 -20341.819,E2 -20341.819} C_VEL
LIN {X 0,Y 221.251,Z 241.917,A -85,B 0,C 180,E1 -20347.3,E2 -20347.3} C_VEL
LIN {X 0,Y 221.059,Z 241.91,A -85,B 0,C 180,E1 -20350.997,E2 -20350.997} C_VEL
LIN {X 0,Y 220.97,Z 241.954,A -85,B 0,C 180,E1 -20354.741,E2 -20354.741} C_VEL
LIN {X 0,Y 220.907,Z 241.941,A -85,B 0,C 180,E1 -20358.551,E2 -20358.551} C_VEL
LIN {X 0,Y 220.89,Z 241.949,A -85,B 0,C 180,E1 -20362.684,E2 -20362.684} C_VEL
LIN {X 0,Y 220.877,Z 241.971,A -85,B 0,C 180,E1 -20367.016,E2 -20367.016} C_VEL
LIN {X 0,Y 220.849,Z 241.96,A -85,B 0,C 180,E1 -20370.344,E2 -20370.344} C_VEL
LIN {X 0,Y 221.775,Z 244.716,A -85,B 0,C 180,E1 -20370.796,E2 -20370.796} C_VEL
LIN {X 0,Y 223.785,Z 246.881,A -85,B 0,C 180,E1 -20371.541,E2 -20371.541} C_VEL
LIN {X 0,Y 224.55,Z 247.672,A -85,B 0,C 180,E1 -20371.816,E2 -20371.816} C_VEL
LIN {X 0,Y 226.571,Z 250.864,A -85,B 0,C 180,E1 -20372.58,E2 -20372.58} C_VEL
LIN {X 0,Y 228.061,Z 252.661,A -85,B 0,C 180,E1 -20373.1,E2 -20373.1} C_VEL
LIN {X 0,Y 230.669,Z 256.174,A -85,B 0,C 180,E1 -20373.999,E2 -20373.999} C_VEL
LIN {X 0,Y 238.839,Z 268.312,A -85,B 0,C 180,E1 -20376.641,E2 -20376.641} C_VEL
LIN {X 0,Y 247.2,Z 282.39,A -85,B 0,C 180,E1 -20379.11,E2 -20379.11} C_VEL
LIN {X 0,Y 252.296,Z 291.953,A -85,B 0,C 180,E1 -20380.521,E2 -20380.521} C_VEL
LIN {X 0,Y 249.512,Z 345.14,A -85,B 0,C 180,E1 -20382.015,E2 -20382.015} C_VEL
LIN {X 0,Y 248.297,Z 358.04,A -85,B 0,C 180,E1 -20382.667,E2 -20382.667} C_VEL
LIN {X 0,Y 246.475,Z 370.236,A -85,B 0,C 180,E1 -20383.581,E2 -20383.581} C_VEL
LIN {X 0,Y 244.022,Z 382.524,A -85,B 0,C 180,E1 -20384.832,E2 -20384.832} C_VEL
LIN {X 0,Y 241.185,Z 394.02,A -85,B 0,C 180,E1 -20386.394,E2 -20386.394} C_VEL
LIN {X 0,Y 237.826,Z 405.107,A -85,B 0,C 180,E1 -20388.328,E2 -20388.328} C_VEL
LIN {X 0,Y 234.526,Z 414.572,A -85,B 0,C 180,E1 -20390.449,E2 -20390.449} C_VEL
LIN {X 0,Y 230.981,Z 423.636,A -85,B 0,C 180,E1 -20393.066,E2 -20393.066} C_VEL
LIN {X 0,Y 227.936,Z 430.829,A -85,B 0,C 180,E1 -20395.759,E2 -20395.759} C_VEL
LIN {X 0,Y 224.917,Z 437.286,A -85,B 0,C 180,E1 -20398.966,E2 -20398.966} C_VEL
LIN {X 0,Y 222.64,Z 441.872,A -85,B 0,C 180,E1 -20402.114,E2 -20402.114} C_VEL
LIN {X 0,Y 220.753,Z 445.204,A -85,B 0,C 180,E1 -20405.554,E2 -20405.554} C_VEL
LIN {X 0,Y 219.79,Z 446.676,A -85,B 0,C 180,E1 -20408.02,E2 -20408.02} C_VEL
LIN {X 0,Y 218.912,Z 447.496,A -85,B 0,C 180,E1 -20411.276,E2 -20411.276} C_VEL
LIN {X 0,Y 218.533,Z 447.032,A -85,B 0,C 180,E1 -20414.755,E2 -20414.755} C_VEL
LIN {X 0,Y 218.468,Z 445.962,A -85,B 0,C 180,E1 -20416.988,E2 -20416.988} C_VEL
LIN {X 0,Y 218.507,Z 444.62,A -85,B 0,C 180,E1 -20418.875,E2 -20418.875} C_VEL
LIN {X 0,Y 218.884,Z 441.768,A -85,B 0,C 180,E1 -20421.694,E2 -20421.694} C_VEL
LIN {X 0,Y 219.482,Z 437.876,A -85,B 0,C 180,E1 -20424.49,E2 -20424.49} C_VEL
LIN {X 0,Y 220.23,Z 432.859,A -85,B 0,C 180,E1 -20427.258,E2 -20427.258} C_VEL
LIN {X 0,Y 221.297,Z 426.517,A -85,B 0,C 180,E1 -20430.002,E2 -20430.002} C_VEL
LIN {X 0,Y 222.811,Z 418.583,A -85,B 0,C 180,E1 -20432.714,E2 -20432.714} C_VEL
LIN {X 0,Y 224.366,Z 410.486,A -85,B 0,C 180,E1 -20434.944,E2 -20434.944} C_VEL
LIN {X 0,Y 226.239,Z 400.586,A -85,B 0,C 180,E1 -20437.14,E2 -20437.14} C_VEL
LIN {X 0,Y 228.116,Z 389.426,A -85,B 0,C 180,E1 -20439.087,E2 -20439.087} C_VEL
LIN {X 0,Y 229.696,Z 378.534,A -85,B 0,C 180,E1 -20440.58,E2 -20440.58} C_VEL
LIN {X 0,Y 230.93,Z 366.514,A -85,B 0,C 180,E1 -20441.856,E2 -20441.856} C_VEL
LIN {X 0,Y 232.116,Z 353.135,A -85,B 0,C 180,E1 -20442.849,E2 -20442.849} C_VEL
LIN {X 0,Y 232.844,Z 339.722,A -85,B 0,C 180,E1 -20443.474,E2 -20443.474} C_VEL
LIN {X 0,Y 235.112,Z 274.125,A -85,B 0,C 180,E1 -20445.413,E2 -20445.413} C_VEL
LIN {X 0,Y 227.925,Z 257.091,A -85,B 0,C 180,E1 -20446.82,E2 -20446.82} C_VEL
LIN {X 0,Y 222.021,Z 244.888,A -85,B 0,C 180,E1 -20447.991,E2 -20447.991} C_VEL
LIN {X 0,Y 220.948,Z 241.962,A -85,B 0,C 180,E1 -20448.248,E2 -20448.248} C_VEL
LIN {X 0,Y 220.863,Z 241.97,A -85,B 0,C 180,E1 -20452.659,E2 -20452.659} C_VEL
LIN {X 0,Y 220.854,Z 241.971,A -85,B 0,C 180,E1 -20456.997,E2 -20456.997} C_VEL
LIN {X 0,Y 220.825,Z 241.97,A -85,B 0,C 180,E1 -20460.76,E2 -20460.76} C_VEL
LIN {X 0,Y 220.799,Z 241.978,A -85,B 0,C 180,E1 -20464.958,E2 -20464.958} C_VEL
LIN {X 0,Y 220.807,Z 241.974,A -85,B 0,C 180,E1 -20467.276,E2 -20467.276} C_VEL
LIN {X 0,Y 220.755,Z 241.976,A -85,B 0,C 180,E1 -20471.959,E2 -20471.959} C_VEL
LIN {X 0,Y 220.759,Z 241.984,A -85,B 0,C 180,E1 -20475.541,E2 -20475.541} C_VEL
LIN {X 0,Y 220.787,Z 241.969,A -85,B 0,C 180,E1 -20480.458,E2 -20480.458} C_VEL
LIN {X 0,Y 220.832,Z 241.963,A -85,B 0,C 180,E1 -20482.794,E2 -20482.794} C_VEL
LIN {X 0,Y 220.818,Z 241.976,A -85,B 0,C 180,E1 -20487.243,E2 -20487.243} C_VEL
LIN {X 0,Y 220.822,Z 241.953,A -85,B 0,C 180,E1 -20491.484,E2 -20491.484} C_VEL
LIN {X 0,Y 220.936,Z 242.133,A -85,B 0,C 180,E1 -20492.879,E2 -20492.879} C_VEL
LIN {X 0,Y 228.13,Z 269.727,A -85,B 0,C 180,E1 -20494.65,E2 -20494.65} C_VEL
LIN {X 0,Y 224.614,Z 346.412,A -85,B 0,C 180,E1 -20498.79,E2 -20498.79} C_VEL
LIN {X 0,Y 223.872,Z 361.26,A -85,B 0,C 180,E1 -20499.991,E2 -20499.991} C_VEL
LIN {X 0,Y 223.007,Z 373.834,A -85,B 0,C 180,E1 -20501.375,E2 -20501.375} C_VEL
LIN {X 0,Y 222.134,Z 385.44,A -85,B 0,C 180,E1 -20502.982,E2 -20502.982} C_VEL
LIN {X 0,Y 221.248,Z 397.298,A -85,B 0,C 180,E1 -20505.043,E2 -20505.043} C_VEL
LIN {X 0,Y 220.454,Z 407.001,A -85,B 0,C 180,E1 -20507.105,E2 -20507.105} C_VEL
LIN {X 0,Y 219.832,Z 416.014,A -85,B 0,C 180,E1 -20509.407,E2 -20509.407} C_VEL
LIN {X 0,Y 219.278,Z 424.796,A -85,B 0,C 180,E1 -20512.171,E2 -20512.171} C_VEL
LIN {X 0,Y 218.911,Z 432.639,A -85,B 0,C 180,E1 -20515.251,E2 -20515.251} C_VEL
LIN {X 0,Y 218.836,Z 438.455,A -85,B 0,C 180,E1 -20518.159,E2 -20518.159} C_VEL
LIN {X 0,Y 218.885,Z 442.758,A -85,B 0,C 180,E1 -20520.919,E2 -20520.919} C_VEL
LIN {X 0,Y 219.337,Z 446.028,A -85,B 0,C 180,E1 -20523.674,E2 -20523.674} C_VEL
LIN {X 0,Y 220.213,Z 448.499,A -85,B 0,C 180,E1 -20526.748,E2 -20526.748} C_VEL
LIN {X 0,Y 219.892,Z 449.14,A -85,B 0,C 180,E1 -20527.77,E2 -20527.77} C_VEL
LIN {X 0,Y 215.685,Z 450.474,A -85,B 0,C 180,E1 -20531.133,E2 -20531.133} C_VEL
LIN {X 0,Y 215.771,Z 450.653,A -85,B 0,C 180,E1 -20532.185,E2 -20532.185} C_VEL
LIN {X 0,Y 218.214,Z 450.681,A -85,B 0,C 180,E1 -20534.931,E2 -20534.931} C_VEL
LIN {X 0,Y 222.175,Z 449.343,A -85,B 0,C 180,E1 -20538.441,E2 -20538.441} C_VEL
LIN {X 0,Y 226.891,Z 446.454,A -85,B 0,C 180,E1 -20541.82,E2 -20541.82} C_VEL
LIN {X 0,Y 232.64,Z 441.965,A -85,B 0,C 180,E1 -20545.02,E2 -20545.02} C_VEL
LIN {X 0,Y 237.451,Z 437.439,A -85,B 0,C 180,E1 -20547.307,E2 -20547.307} C_VEL
LIN {X 0,Y 243.614,Z 430.772,A -85,B 0,C 180,E1 -20549.844,E2 -20549.844} C_VEL
LIN {X 0,Y 249.551,Z 423.53,A -85,B 0,C 180,E1 -20551.921,E2 -20551.921} C_VEL
LIN {X 0,Y 255.863,Z 414.789,A -85,B 0,C 180,E1 -20553.898,E2 -20553.898} C_VEL
LIN {X 0,Y 262.133,Z 404.758,A -85,B 0,C 180,E1 -20555.671,E2 -20555.671} C_VEL
LIN {X 0,Y 267.94,Z 394.212,A -85,B 0,C 180,E1 -20557.105,E2 -20557.105} C_VEL
LIN {X 0,Y 273.329,Z 382.735,A -85,B 0,C 180,E1 -20558.339,E2 -20558.339} C_VEL
LIN {X 0,Y 278.239,Z 370.304,A -85,B 0,C 180,E1 -20559.39,E2 -20559.39} C_VEL
LIN {X 0,Y 282.764,Z 355.954,A -85,B 0,C 180,E1 -20560.257,E2 -20560.257} C_VEL
LIN {X 0,Y 287.415,Z 336.962,A -85,B 0,C 180,E1 -20561.145,E2 -20561.145} C_VEL
LIN {X 0,Y 287.12,Z 336.406,A -85,B 0,C 180,E1 -20562.053,E2 -20562.053} C_VEL
LIN {X 0,Y 286.707,Z 336.636,A -85,B 0,C 180,E1 -20564.323,E2 -20564.323} C_VEL
LIN {X 0,Y 286.682,Z 337.491,A -85,B 0,C 180,E1 -20565.407,E2 -20565.407} C_VEL
LIN {X 0,Y 286.796,Z 340.534,A -85,B 0,C 180,E1 -20567.305,E2 -20567.305} C_VEL
LIN {X 0,Y 281.246,Z 362.874,A -85,B 0,C 180,E1 -20568.316,E2 -20568.316} C_VEL
LIN {X 0,Y 276.438,Z 377.286,A -85,B 0,C 180,E1 -20569.105,E2 -20569.105} C_VEL
LIN {X 0,Y 270.311,Z 391.98,A -85,B 0,C 180,E1 -20570.188,E2 -20570.188} C_VEL
LIN {X 0,Y 264.424,Z 403.847,A -85,B 0,C 180,E1 -20571.346,E2 -20571.346} C_VEL
LIN {X 0,Y 257.12,Z 416.589,A -85,B 0,C 180,E1 -20573.032,E2 -20573.032} C_VEL
LIN {X 0,Y 250.255,Z 427.053,A -85,B 0,C 180,E1 -20574.849,E2 -20574.849} C_VEL
LIN {X 0,Y 242.99,Z 437.017,A -85,B 0,C 180,E1 -20577.157,E2 -20577.157} C_VEL
LIN {X 0,Y 236.384,Z 445.087,A -85,B 0,C 180,E1 -20579.638,E2 -20579.638} C_VEL
LIN {X 0,Y 231.277,Z 450.767,A -85,B 0,C 180,E1 -20581.898,E2 -20581.898} C_VEL
LIN {X 0,Y 225.292,Z 456.76,A -85,B 0,C 180,E1 -20585.092,E2 -20585.092} C_VEL
LIN {X 0,Y 221.564,Z 460.154,A -85,B 0,C 180,E1 -20587.625,E2 -20587.625} C_VEL
LIN {X 0,Y 217.562,Z 463.378,A -85,B 0,C 180,E1 -20591.151,E2 -20591.151} C_VEL
LIN {X 0,Y 214.453,Z 465.121,A -85,B 0,C 180,E1 -20594.799,E2 -20594.799} C_VEL
LIN {X 0,Y 212.679,Z 465.417,A -85,B 0,C 180,E1 -20598.562,E2 -20598.562} C_VEL
LIN {X 0,Y 211.91,Z 464.275,A -85,B 0,C 180,E1 -20602.375,E2 -20602.375} C_VEL
LIN {X 0,Y 211.927,Z 462.175,A -85,B 0,C 180,E1 -20605.59,E2 -20605.59} C_VEL
LIN {X 0,Y 211.81,Z 464.289,A -85,B 0,C 180,E1 -20608.096,E2 -20608.096} C_VEL
LIN {X 0,Y 211.857,Z 465.397,A -85,B 0,C 180,E1 -20609.998,E2 -20609.998} C_VEL
LIN {X 0,Y 211.742,Z 466.058,A -85,B 0,C 180,E1 -20611.9,E2 -20611.9} C_VEL
LIN {X 0,Y 211.565,Z 466.202,A -85,B 0,C 180,E1 -20615.717,E2 -20615.717} C_VEL
LIN {X 0,Y 211.647,Z 465.66,A -85,B 0,C 180,E1 -20617.631,E2 -20617.631} C_VEL
LIN {X 0,Y 212.483,Z 463.375,A -85,B 0,C 180,E1 -20621.444,E2 -20621.444} C_VEL
LIN {X 0,Y 213.624,Z 460.577,A -85,B 0,C 180,E1 -20624.283,E2 -20624.283} C_VEL
LIN {X 0,Y 215.431,Z 456.778,A -85,B 0,C 180,E1 -20627.072,E2 -20627.072} C_VEL
LIN {X 0,Y 217.629,Z 451.866,A -85,B 0,C 180,E1 -20629.819,E2 -20629.819} C_VEL
LIN {X 0,Y 220.249,Z 445.702,A -85,B 0,C 180,E1 -20632.512,E2 -20632.512} C_VEL
LIN {X 0,Y 223.521,Z 438.035,A -85,B 0,C 180,E1 -20635.115,E2 -20635.115} C_VEL
LIN {X 0,Y 227.389,Z 428.447,A -85,B 0,C 180,E1 -20637.618,E2 -20637.618} C_VEL
LIN {X 0,Y 230.929,Z 418.545,A -85,B 0,C 180,E1 -20639.638,E2 -20639.638} C_VEL
LIN {X 0,Y 234.325,Z 407.361,A -85,B 0,C 180,E1 -20641.405,E2 -20641.405} C_VEL
LIN {X 0,Y 237.291,Z 396.408,A -85,B 0,C 180,E1 -20642.717,E2 -20642.717} C_VEL
LIN {X 0,Y 239.986,Z 384.206,A -85,B 0,C 180,E1 -20643.806,E2 -20643.806} C_VEL
LIN {X 0,Y 241.992,Z 371.361,A -85,B 0,C 180,E1 -20644.618,E2 -20644.618} C_VEL
LIN {X 0,Y 243.235,Z 357.901,A -85,B 0,C 180,E1 -20645.172,E2 -20645.172} C_VEL
LIN {X 0,Y 245.339,Z 315.441,A -85,B 0,C 180,E1 -20646.395,E2 -20646.395} C_VEL
LIN {X 0,Y 242.532,Z 290.727,A -85,B 0,C 180,E1 -20647.984,E2 -20647.984} C_VEL
LIN {X 0,Y 238.862,Z 280.065,A -85,B 0,C 180,E1 -20649.269,E2 -20649.269} C_VEL
LIN {X 0,Y 231.718,Z 268.581,A -85,B 0,C 180,E1 -20651.56,E2 -20651.56} C_VEL
LIN {X 0,Y 226.461,Z 260.961,A -85,B 0,C 180,E1 -20653.377,E2 -20653.377} C_VEL
LIN {X 0,Y 223.463,Z 256.797,A -85,B 0,C 180,E1 -20654.474,E2 -20654.474} C_VEL
LIN {X 0,Y 220.463,Z 252.675,A -85,B 0,C 180,E1 -20655.627,E2 -20655.627} C_VEL
LIN {X 0,Y 218.107,Z 249.765,A -85,B 0,C 180,E1 -20656.564,E2 -20656.564} C_VEL
LIN {X 0,Y 217.336,Z 248.209,A -85,B 0,C 180,E1 -20656.912,E2 -20656.912} C_VEL
LIN {X 0,Y 215.011,Z 246.167,A -85,B 0,C 180,E1 -20657.848,E2 -20657.848} C_VEL
LIN {X 0,Y 213.821,Z 243.603,A -85,B 0,C 180,E1 -20658.43,E2 -20658.43} C_VEL
LIN {X 0,Y 213.698,Z 242.842,A -85,B 0,C 180,E1 -20658.558,E2 -20658.558} C_VEL
LIN {X 0,Y 213.734,Z 242.831,A -85,B 0,C 180,E1 -20663.71,E2 -20663.71} C_VEL
LIN {X 0,Y 213.751,Z 242.844,A -85,B 0,C 180,E1 -20668.26,E2 -20668.26} C_VEL
LIN {X 0,Y 213.776,Z 242.83,A -85,B 0,C 180,E1 -20672.597,E2 -20672.597} C_VEL
LIN {X 0,Y 213.791,Z 242.813,A -85,B 0,C 180,E1 -20676.986,E2 -20676.986} C_VEL
LIN {X 0,Y 213.878,Z 242.836,A -85,B 0,C 180,E1 -20682.798,E2 -20682.798} C_VEL
LIN {X 0,Y 213.917,Z 242.796,A -85,B 0,C 180,E1 -20686.705,E2 -20686.705} C_VEL
LIN {X 0,Y 214.125,Z 242.813,A -85,B 0,C 180,E1 -20690.555,E2 -20690.555} C_VEL
LIN {X 0,Y 214.068,Z 242.775,A -85,B 0,C 180,E1 -20694.348,E2 -20694.348} C_VEL
LIN {X 0,Y 214.4,Z 242.772,A -85,B 0,C 180,E1 -20698.122,E2 -20698.122} C_VEL
LIN {X 0,Y 214.505,Z 242.751,A -85,B 0,C 180,E1 -20700,E2 -20700} C_VEL
LIN {X 0,Y 214.401,Z 242.736,A -85,B 0,C 180,E1 -20701.879,E2 -20701.879} C_VEL
LIN {X 0,Y 214.19,Z 242.793,A -85,B 0,C 180,E1 -20707.542,E2 -20707.542} C_VEL
LIN {X 0,Y 213.99,Z 242.792,A -85,B 0,C 180,E1 -20711.365,E2 -20711.365} C_VEL
LIN {X 0,Y 213.906,Z 242.826,A -85,B 0,C 180,E1 -20715.239,E2 -20715.239} C_VEL
LIN {X 0,Y 213.826,Z 242.829,A -85,B 0,C 180,E1 -20719.189,E2 -20719.189} C_VEL
LIN {X 0,Y 213.841,Z 242.823,A -85,B 0,C 180,E1 -20723.228,E2 -20723.228} C_VEL
LIN {X 0,Y 213.809,Z 242.982,A -85,B 0,C 180,E1 -20727.938,E2 -20727.938} C_VEL
LIN {X 0,Y 214.645,Z 245.428,A -85,B 0,C 180,E1 -20728.385,E2 -20728.385} C_VEL
LIN {X 0,Y 216.446,Z 247.53,A -85,B 0,C 180,E1 -20729.148,E2 -20729.148} C_VEL
LIN {X 0,Y 217.552,Z 248.365,A -85,B 0,C 180,E1 -20729.579,E2 -20729.579} C_VEL
LIN {X 0,Y 219.507,Z 251.633,A -85,B 0,C 180,E1 -20730.414,E2 -20730.414} C_VEL
LIN {X 0,Y 221.4,Z 253.744,A -85,B 0,C 180,E1 -20731.139,E2 -20731.139} C_VEL
LIN {X 0,Y 224.213,Z 257.516,A -85,B 0,C 180,E1 -20732.2,E2 -20732.2} C_VEL
LIN {X 0,Y 227.327,Z 261.883,A -85,B 0,C 180,E1 -20733.327,E2 -20733.327} C_VEL
LIN {X 0,Y 235.263,Z 273.962,A -85,B 0,C 180,E1 -20736.005,E2 -20736.005} C_VEL
LIN {X 0,Y 242.862,Z 286.958,A -85,B 0,C 180,E1 -20738.344,E2 -20738.344} C_VEL
LIN {X 0,Y 246.884,Z 294.544,A -85,B 0,C 180,E1 -20739.517,E2 -20739.517} C_VEL
LIN {X 0,Y 244.16,Z 344.303,A -85,B 0,C 180,E1 -20740.923,E2 -20740.923} C_VEL
LIN {X 0,Y 242.879,Z 357.685,A -85,B 0,C 180,E1 -20741.581,E2 -20741.581} C_VEL
LIN {X 0,Y 241.156,Z 369.078,A -85,B 0,C 180,E1 -20742.414,E2 -20742.414} C_VEL
LIN {X 0,Y 238.858,Z 380.676,A -85,B 0,C 180,E1 -20743.571,E2 -20743.571} C_VEL
LIN {X 0,Y 236.105,Z 391.784,A -85,B 0,C 180,E1 -20745.016,E2 -20745.016} C_VEL
LIN {X 0,Y 233.077,Z 401.921,A -85,B 0,C 180,E1 -20746.69,E2 -20746.69} C_VEL
LIN {X 0,Y 229.505,Z 412.04,A -85,B 0,C 180,E1 -20748.826,E2 -20748.826} C_VEL
LIN {X 0,Y 226.169,Z 420.534,A -85,B 0,C 180,E1 -20751.111,E2 -20751.111} C_VEL
LIN {X 0,Y 222.858,Z 428.229,A -85,B 0,C 180,E1 -20753.754,E2 -20753.754} C_VEL
LIN {X 0,Y 219.939,Z 434.414,A -85,B 0,C 180,E1 -20756.502,E2 -20756.502} C_VEL
LIN {X 0,Y 217.024,Z 440.113,A -85,B 0,C 180,E1 -20759.874,E2 -20759.874} C_VEL
LIN {X 0,Y 215.093,Z 443.603,A -85,B 0,C 180,E1 -20762.78,E2 -20762.78} C_VEL
LIN {X 0,Y 214.032,Z 445.301,A -85,B 0,C 180,E1 -20764.733,E2 -20764.733} C_VEL
LIN {X 0,Y 212.813,Z 447.012,A -85,B 0,C 180,E1 -20767.622,E2 -20767.622} C_VEL
LIN {X 0,Y 211.937,Z 447.795,A -85,B 0,C 180,E1 -20770.636,E2 -20770.636} C_VEL
LIN {X 0,Y 211.628,Z 447.765,A -85,B 0,C 180,E1 -20772.612,E2 -20772.612} C_VEL
LIN {X 0,Y 211.464,Z 447.336,A -85,B 0,C 180,E1 -20774.583,E2 -20774.583} C_VEL
LIN {X 0,Y 211.364,Z 446.459,A -85,B 0,C 180,E1 -20776.543,E2 -20776.543} C_VEL
LIN {X 0,Y 211.385,Z 445.165,A -85,B 0,C 180,E1 -20778.495,E2 -20778.495} C_VEL
LIN {X 0,Y 211.734,Z 442.415,A -85,B 0,C 180,E1 -20781.412,E2 -20781.412} C_VEL
LIN {X 0,Y 212.333,Z 438.629,A -85,B 0,C 180,E1 -20784.303,E2 -20784.303} C_VEL
LIN {X 0,Y 213.091,Z 433.726,A -85,B 0,C 180,E1 -20787.166,E2 -20787.166} C_VEL
LIN {X 0,Y 214.178,Z 427.553,A -85,B 0,C 180,E1 -20790.002,E2 -20790.002} C_VEL
LIN {X 0,Y 215.707,Z 419.794,A -85,B 0,C 180,E1 -20792.803,E2 -20792.803} C_VEL
LIN {X 0,Y 217.295,Z 411.869,A -85,B 0,C 180,E1 -20795.105,E2 -20795.105} C_VEL
LIN {X 0,Y 219.138,Z 402.225,A -85,B 0,C 180,E1 -20797.372,E2 -20797.372} C_VEL
LIN {X 0,Y 221.048,Z 391.816,A -85,B 0,C 180,E1 -20799.315,E2 -20799.315} C_VEL
LIN {X 0,Y 222.732,Z 380.917,A -85,B 0,C 180,E1 -20800.915,E2 -20800.915} C_VEL
LIN {X 0,Y 224.116,Z 368.479,A -85,B 0,C 180,E1 -20802.337,E2 -20802.337} C_VEL
LIN {X 0,Y 225.385,Z 355.818,A -85,B 0,C 180,E1 -20803.355,E2 -20803.355} C_VEL
LIN {X 0,Y 226.184,Z 342.625,A -85,B 0,C 180,E1 -20804.051,E2 -20804.051} C_VEL
LIN {X 0,Y 228.587,Z 275.782,A -85,B 0,C 180,E1 -20806.097,E2 -20806.097} C_VEL
LIN {X 0,Y 221.065,Z 258.048,A -85,B 0,C 180,E1 -20807.642,E2 -20807.642} C_VEL
LIN {X 0,Y 214.779,Z 245.519,A -85,B 0,C 180,E1 -20808.947,E2 -20808.947} C_VEL
LIN {X 0,Y 213.842,Z 242.848,A -85,B 0,C 180,E1 -20809.189,E2 -20809.189} C_VEL
LIN {X 0,Y 213.801,Z 242.85,A -85,B 0,C 180,E1 -20813.234,E2 -20813.234} C_VEL
LIN {X 0,Y 213.791,Z 242.851,A -85,B 0,C 180,E1 -20817.428,E2 -20817.428} C_VEL
LIN {X 0,Y 213.765,Z 242.852,A -85,B 0,C 180,E1 -20821.74,E2 -20821.74} C_VEL
LIN {X 0,Y 213.748,Z 242.851,A -85,B 0,C 180,E1 -20826.29,E2 -20826.29} C_VEL
LIN {X 0,Y 213.704,Z 242.861,A -85,B 0,C 180,E1 -20831.13,E2 -20831.13} C_VEL
LIN {X 0,Y 213.708,Z 242.853,A -85,B 0,C 180,E1 -20833.681,E2 -20833.681} C_VEL
LIN {X 0,Y 213.707,Z 242.862,A -85,B 0,C 180,E1 -20836.346,E2 -20836.346} C_VEL
LIN {X 0,Y 213.707,Z 242.846,A -85,B 0,C 180,E1 -20841.329,E2 -20841.329} C_VEL
LIN {X 0,Y 213.76,Z 242.855,A -85,B 0,C 180,E1 -20846.018,E2 -20846.018} C_VEL
LIN {X 0,Y 213.762,Z 242.839,A -85,B 0,C 180,E1 -20850.45,E2 -20850.45} C_VEL
LIN {X 0,Y 213.834,Z 242.825,A -85,B 0,C 180,E1 -20852.604,E2 -20852.604} C_VEL
LIN {X 0,Y 221.014,Z 270.862,A -85,B 0,C 180,E1 -20854.483,E2 -20854.483} C_VEL
LIN {X 0,Y 217.498,Z 347.342,A -85,B 0,C 180,E1 -20858.807,E2 -20858.807} C_VEL
LIN {X 0,Y 216.777,Z 361.284,A -85,B 0,C 180,E1 -20859.984,E2 -20859.984} C_VEL
LIN {X 0,Y 215.848,Z 374.44,A -85,B 0,C 180,E1 -20861.49,E2 -20861.49} C_VEL
LIN {X 0,Y 214.993,Z 385.832,A -85,B 0,C 180,E1 -20863.134,E2 -20863.134} C_VEL
LIN {X 0,Y 214.131,Z 397.676,A -85,B 0,C 180,E1 -20865.264,E2 -20865.264} C_VEL
LIN {X 0,Y 213.222,Z 408.312,A -85,B 0,C 180,E1 -20867.628,E2 -20867.628} C_VEL
LIN {X 0,Y 212.617,Z 417.095,A -85,B 0,C 180,E1 -20870.006,E2 -20870.006} C_VEL
LIN {X 0,Y 212.149,Z 425.735,A -85,B 0,C 180,E1 -20872.864,E2 -20872.864} C_VEL
LIN {X 0,Y 211.859,Z 432.675,A -85,B 0,C 180,E1 -20875.705,E2 -20875.705} C_VEL
LIN {X 0,Y 211.784,Z 437.454,A -85,B 0,C 180,E1 -20878.098,E2 -20878.098} C_VEL
LIN {X 0,Y 211.818,Z 442.037,A -85,B 0,C 180,E1 -20880.95,E2 -20880.95} C_VEL
LIN {X 0,Y 212.283,Z 445.586,A -85,B 0,C 180,E1 -20883.796,E2 -20883.796} C_VEL
LIN {X 0,Y 213.383,Z 448.852,A -85,B 0,C 180,E1 -20887.57,E2 -20887.57} C_VEL
LIN {X 0,Y 215.061,Z 450.529,A -85,B 0,C 180,E1 -20891.307,E2 -20891.307} C_VEL
LIN {X 0,Y 215.771,Z 450.653,A -85,B 0,C 180,E1 -20892.185,E2 -20892.185} C_VEL
LIN {X 0,Y 216.458,Z 450.853,A -85,B 0,C 180,E1 -20893.738,E2 -20893.738} C_VEL
LIN {X 0,Y 216.112,Z 450.783,A -85,B 0,C 180,E1 -20896.361,E2 -20896.361} C_VEL
LIN {X 0,Y 216.172,Z 450.248,A -85,B 0,C 180,E1 -20898.983,E2 -20898.983} C_VEL
LIN {X 0,Y 217.471,Z 449.487,A -85,B 0,C 180,E1 -20900.492,E2 -20900.492} C_VEL
LIN {X 0,Y 220.46,Z 447.928,A -85,B 0,C 180,E1 -20902.491,E2 -20902.491} C_VEL
LIN {X 0,Y 224.859,Z 445.065,A -85,B 0,C 180,E1 -20904.957,E2 -20904.957} C_VEL
LIN {X 0,Y 229.703,Z 441.291,A -85,B 0,C 180,E1 -20907.318,E2 -20907.318} C_VEL
LIN {X 0,Y 235.714,Z 435.878,A -85,B 0,C 180,E1 -20909.815,E2 -20909.815} C_VEL
LIN {X 0,Y 241.351,Z 430.053,A -85,B 0,C 180,E1 -20911.869,E2 -20911.869} C_VEL
LIN {X 0,Y 248.149,Z 422.114,A -85,B 0,C 180,E1 -20914.011,E2 -20914.011} C_VEL
LIN {X 0,Y 254.755,Z 413.211,A -85,B 0,C 180,E1 -20915.89,E2 -20915.89} C_VEL
LIN {X 0,Y 260.548,Z 404.372,A -85,B 0,C 180,E1 -20917.366,E2 -20917.366} C_VEL
LIN {X 0,Y 267.287,Z 392.538,A -85,B 0,C 180,E1 -20918.885,E2 -20918.885} C_VEL
LIN {X 0,Y 273.58,Z 379.3,A -85,B 0,C 180,E1 -20920.198,E2 -20920.198} C_VEL
LIN {X 0,Y 278.583,Z 366.455,A -85,B 0,C 180,E1 -20921.133,E2 -20921.133} C_VEL
LIN {X 0,Y 282.947,Z 352.118,A -85,B 0,C 180,E1 -20921.906,E2 -20921.906} C_VEL
LIN {X 0,Y 285.202,Z 343.229,A -85,B 0,C 180,E1 -20922.329,E2 -20922.329} C_VEL
LIN {X 0,Y 284.872,Z 343.546,A -85,B 0,C 180,E1 -20924.43,E2 -20924.43} C_VEL
LIN {X 0,Y 284.754,Z 344.803,A -85,B 0,C 180,E1 -20925.494,E2 -20925.494} C_VEL
LIN {X 0,Y 284.737,Z 345.65,A -85,B 0,C 180,E1 -20926.074,E2 -20926.074} C_VEL
LIN {X 0,Y 279.921,Z 363.612,A -85,B 0,C 180,E1 -20926.895,E2 -20926.895} C_VEL
LIN {X 0,Y 274.49,Z 378.746,A -85,B 0,C 180,E1 -20927.719,E2 -20927.719} C_VEL
LIN {X 0,Y 268.685,Z 391.738,A -85,B 0,C 180,E1 -20928.663,E2 -20928.663} C_VEL
LIN {X 0,Y 262.526,Z 403.492,A -85,B 0,C 180,E1 -20929.769,E2 -20929.769} C_VEL
LIN {X 0,Y 255.49,Z 415.13,A -85,B 0,C 180,E1 -20931.257,E2 -20931.257} C_VEL
LIN {X 0,Y 249.423,Z 424.045,A -85,B 0,C 180,E1 -20932.711,E2 -20932.711} C_VEL
LIN {X 0,Y 242.57,Z 433.098,A -85,B 0,C 180,E1 -20934.585,E2 -20934.585} C_VEL
LIN {X 0,Y 235.224,Z 441.737,A -85,B 0,C 180,E1 -20936.955,E2 -20936.955} C_VEL
LIN {X 0,Y 228.607,Z 448.76,A -85,B 0,C 180,E1 -20939.517,E2 -20939.517} C_VEL
LIN {X 0,Y 222.546,Z 454.543,A -85,B 0,C 180,E1 -20942.345,E2 -20942.345} C_VEL
LIN {X 0,Y 217.502,Z 458.741,A -85,B 0,C 180,E1 -20945.159,E2 -20945.159} C_VEL
LIN {X 0,Y 212.832,Z 462.23,A -85,B 0,C 180,E1 -20948.699,E2 -20948.699} C_VEL
LIN {X 0,Y 209.065,Z 464.311,A -85,B 0,C 180,E1 -20952.387,E2 -20952.387} C_VEL
LIN {X 0,Y 206.551,Z 464.997,A -85,B 0,C 180,E1 -20956.219,E2 -20956.219} C_VEL
LIN {X 0,Y 205.205,Z 464.236,A -85,B 0,C 180,E1 -20960.138,E2 -20960.138} C_VEL
LIN {X 0,Y 204.9,Z 462.005,A -85,B 0,C 180,E1 -20964.092,E2 -20964.092} C_VEL
LIN {X 0,Y 204.917,Z 461.301,A -85,B 0,C 180,E1 -20965.063,E2 -20965.063} C_VEL
LIN {X 0,Y 204.746,Z 463.844,A -85,B 0,C 180,E1 -20968.031,E2 -20968.031} C_VEL
LIN {X 0,Y 204.785,Z 465.006,A -85,B 0,C 180,E1 -20969.998,E2 -20969.998} C_VEL
LIN {X 0,Y 204.644,Z 465.699,A -85,B 0,C 180,E1 -20971.966,E2 -20971.966} C_VEL
LIN {X 0,Y 204.485,Z 465.901,A -85,B 0,C 180,E1 -20975.916,E2 -20975.916} C_VEL
LIN {X 0,Y 204.603,Z 465.415,A -85,B 0,C 180,E1 -20977.895,E2 -20977.895} C_VEL
LIN {X 0,Y 205.488,Z 463.194,A -85,B 0,C 180,E1 -20981.839,E2 -20981.839} C_VEL
LIN {X 0,Y 206.712,Z 460.461,A -85,B 0,C 180,E1 -20984.771,E2 -20984.771} C_VEL
LIN {X 0,Y 208.628,Z 456.731,A -85,B 0,C 180,E1 -20987.646,E2 -20987.646} C_VEL
LIN {X 0,Y 210.955,Z 451.892,A -85,B 0,C 180,E1 -20990.473,E2 -20990.473} C_VEL
LIN {X 0,Y 213.698,Z 445.809,A -85,B 0,C 180,E1 -20993.242,E2 -20993.242} C_VEL
LIN {X 0,Y 217.132,Z 438.269,A -85,B 0,C 180,E1 -20995.908,E2 -20995.908} C_VEL
LIN {X 0,Y 221.133,Z 428.805,A -85,B 0,C 180,E1 -20998.469,E2 -20998.469} C_VEL
LIN {X 0,Y 224.822,Z 419.053,A -85,B 0,C 180,E1 -21000.527,E2 -21000.527} C_VEL
LIN {X 0,Y 228.335,Z 408.125,A -85,B 0,C 180,E1 -21002.327,E2 -21002.327} C_VEL
LIN {X 0,Y 231.816,Z 395.711,A -85,B 0,C 180,E1 -21003.851,E2 -21003.851} C_VEL
LIN {X 0,Y 234.665,Z 383.332,A -85,B 0,C 180,E1 -21004.942,E2 -21004.942} C_VEL
LIN {X 0,Y 236.606,Z 371.169,A -85,B 0,C 180,E1 -21005.72,E2 -21005.72} C_VEL
LIN {X 0,Y 237.845,Z 358.275,A -85,B 0,C 180,E1 -21006.269,E2 -21006.269} C_VEL
LIN {X 0,Y 240.047,Z 316.245,A -85,B 0,C 180,E1 -21007.5,E2 -21007.5} C_VEL
LIN {X 0,Y 237.483,Z 293.265,A -85,B 0,C 180,E1 -21009.039,E2 -21009.039} C_VEL
LIN {X 0,Y 234.471,Z 284.337,A -85,B 0,C 180,E1 -21010.152,E2 -21010.152} C_VEL
LIN {X 0,Y 227.941,Z 273.695,A -85,B 0,C 180,E1 -21012.353,E2 -21012.353} C_VEL
LIN {X 0,Y 222.664,Z 265.933,A -85,B 0,C 180,E1 -21014.265,E2 -21014.265} C_VEL
LIN {X 0,Y 219.481,Z 261.546,A -85,B 0,C 180,E1 -21015.486,E2 -21015.486} C_VEL
LIN {X 0,Y 217.227,Z 258.374,A -85,B 0,C 180,E1 -21016.403,E2 -21016.403} C_VEL
LIN {X 0,Y 214.635,Z 254.847,A -85,B 0,C 180,E1 -21017.5,E2 -21017.5} C_VEL
LIN {X 0,Y 213.225,Z 253.294,A -85,B 0,C 180,E1 -21018.1,E2 -21018.1} C_VEL
LIN {X 0,Y 211.141,Z 250.461,A -85,B 0,C 180,E1 -21019.049,E2 -21019.049} C_VEL
LIN {X 0,Y 210.562,Z 249.218,A -85,B 0,C 180,E1 -21019.347,E2 -21019.347} C_VEL
LIN {X 0,Y 208.211,Z 247.375,A -85,B 0,C 180,E1 -21020.401,E2 -21020.401} C_VEL
LIN {X 0,Y 206.976,Z 245.172,A -85,B 0,C 180,E1 -21021.054,E2 -21021.054} C_VEL
LIN {X 0,Y 206.673,Z 243.739,A -85,B 0,C 180,E1 -21021.309,E2 -21021.309} C_VEL
LIN {X 0,Y 206.692,Z 243.707,A -85,B 0,C 180,E1 -21024.688,E2 -21024.688} C_VEL
LIN {X 0,Y 206.687,Z 243.706,A -85,B 0,C 180,E1 -21029.333,E2 -21029.333} C_VEL
LIN {X 0,Y 206.695,Z 243.729,A -85,B 0,C 180,E1 -21033.767,E2 -21033.767} C_VEL
LIN {X 0,Y 206.708,Z 243.691,A -85,B 0,C 180,E1 -21038.038,E2 -21038.038} C_VEL
LIN {X 0,Y 206.813,Z 243.721,A -85,B 0,C 180,E1 -21042.192,E2 -21042.192} C_VEL
LIN {X 0,Y 206.857,Z 243.673,A -85,B 0,C 180,E1 -21046.242,E2 -21046.242} C_VEL
LIN {X 0,Y 207.07,Z 243.692,A -85,B 0,C 180,E1 -21050.23,E2 -21050.23} C_VEL
LIN {X 0,Y 207.031,Z 243.652,A -85,B 0,C 180,E1 -21054.155,E2 -21054.155} C_VEL
LIN {X 0,Y 207.339,Z 243.651,A -85,B 0,C 180,E1 -21058.058,E2 -21058.058} C_VEL
LIN {X 0,Y 207.473,Z 243.625,A -85,B 0,C 180,E1 -21060,E2 -21060} C_VEL
LIN {X 0,Y 207.341,Z 243.614,A -85,B 0,C 180,E1 -21061.943,E2 -21061.943} C_VEL
LIN {X 0,Y 207.133,Z 243.668,A -85,B 0,C 180,E1 -21067.801,E2 -21067.801} C_VEL
LIN {X 0,Y 206.913,Z 243.676,A -85,B 0,C 180,E1 -21071.76,E2 -21071.76} C_VEL
LIN {X 0,Y 206.839,Z 243.697,A -85,B 0,C 180,E1 -21075.773,E2 -21075.773} C_VEL
LIN {X 0,Y 206.773,Z 243.718,A -85,B 0,C 180,E1 -21079.871,E2 -21079.871} C_VEL
LIN {X 0,Y 206.757,Z 243.704,A -85,B 0,C 180,E1 -21084.074,E2 -21084.074} C_VEL
LIN {X 0,Y 206.756,Z 243.711,A -85,B 0,C 180,E1 -21085.145,E2 -21085.145} C_VEL
LIN {X 0,Y 207.635,Z 246.365,A -85,B 0,C 180,E1 -21085.702,E2 -21085.702} C_VEL
LIN {X 0,Y 209.643,Z 248.612,A -85,B 0,C 180,E1 -21086.658,E2 -21086.658} C_VEL
LIN {X 0,Y 210.818,Z 249.578,A -85,B 0,C 180,E1 -21087.179,E2 -21087.179} C_VEL
LIN {X 0,Y 212.729,Z 252.66,A -85,B 0,C 180,E1 -21088.086,E2 -21088.086} C_VEL
LIN {X 0,Y 214.722,Z 254.798,A -85,B 0,C 180,E1 -21088.935,E2 -21088.935} C_VEL
LIN {X 0,Y 217.406,Z 258.489,A -85,B 0,C 180,E1 -21090.071,E2 -21090.071} C_VEL
LIN {X 0,Y 221.877,Z 264.713,A -85,B 0,C 180,E1 -21091.844,E2 -21091.844} C_VEL
LIN {X 0,Y 226.904,Z 272.004,A -85,B 0,C 180,E1 -21093.685,E2 -21093.685} C_VEL
LIN {X 0,Y 233.581,Z 282.684,A -85,B 0,C 180,E1 -21095.962,E2 -21095.962} C_VEL
LIN {X 0,Y 241.2,Z 296.404,A -85,B 0,C 180,E1 -21098.353,E2 -21098.353} C_VEL
LIN {X 0,Y 241.575,Z 297.205,A -85,B 0,C 180,E1 -21098.47,E2 -21098.47} C_VEL
LIN {X 0,Y 238.802,Z 344.946,A -85,B 0,C 180,E1 -21099.832,E2 -21099.832} C_VEL
LIN {X 0,Y 237.451,Z 358.271,A -85,B 0,C 180,E1 -21100.502,E2 -21100.502} C_VEL
LIN {X 0,Y 235.527,Z 370.357,A -85,B 0,C 180,E1 -21101.42,E2 -21101.42} C_VEL
LIN {X 0,Y 232.946,Z 382.4,A -85,B 0,C 180,E1 -21102.662,E2 -21102.662} C_VEL
LIN {X 0,Y 230.097,Z 393.231,A -85,B 0,C 180,E1 -21104.132,E2 -21104.132} C_VEL
LIN {X 0,Y 226.538,Z 404.293,A -85,B 0,C 180,E1 -21106.074,E2 -21106.074} C_VEL
LIN {X 0,Y 223.254,Z 413.064,A -85,B 0,C 180,E1 -21108.017,E2 -21108.017} C_VEL
LIN {X 0,Y 219.9,Z 421.168,A -85,B 0,C 180,E1 -21110.271,E2 -21110.271} C_VEL
LIN {X 0,Y 216.875,Z 427.819,A -85,B 0,C 180,E1 -21112.586,E2 -21112.586} C_VEL
LIN {X 0,Y 213.947,Z 433.807,A -85,B 0,C 180,E1 -21115.21,E2 -21115.21} C_VEL
LIN {X 0,Y 211.42,Z 438.552,A -85,B 0,C 180,E1 -21117.871,E2 -21117.871} C_VEL
LIN {X 0,Y 209.098,Z 442.614,A -85,B 0,C 180,E1 -21120.915,E2 -21120.915} C_VEL
LIN {X 0,Y 207.331,Z 445.401,A -85,B 0,C 180,E1 -21123.856,E2 -21123.856} C_VEL
LIN {X 0,Y 205.867,Z 447.344,A -85,B 0,C 180,E1 -21127.184,E2 -21127.184} C_VEL
LIN {X 0,Y 204.99,Z 448.094,A -85,B 0,C 180,E1 -21129.952,E2 -21129.952} C_VEL
LIN {X 0,Y 204.624,Z 448.113,A -85,B 0,C 180,E1 -21131.997,E2 -21131.997} C_VEL
LIN {X 0,Y 204.379,Z 447.657,A -85,B 0,C 180,E1 -21134.334,E2 -21134.334} C_VEL
LIN {X 0,Y 204.265,Z 445.707,A -85,B 0,C 180,E1 -21138.089,E2 -21138.089} C_VEL
LIN {X 0,Y 204.581,Z 443.056,A -85,B 0,C 180,E1 -21141.109,E2 -21141.109} C_VEL
LIN {X 0,Y 205.19,Z 439.374,A -85,B 0,C 180,E1 -21144.104,E2 -21144.104} C_VEL
LIN {X 0,Y 205.957,Z 434.581,A -85,B 0,C 180,E1 -21147.068,E2 -21147.068} C_VEL
LIN {X 0,Y 207.06,Z 428.529,A -85,B 0,C 180,E1 -21150.002,E2 -21150.002} C_VEL
LIN {X 0,Y 208.606,Z 420.982,A -85,B 0,C 180,E1 -21152.899,E2 -21152.899} C_VEL
LIN {X 0,Y 210.547,Z 411.482,A -85,B 0,C 180,E1 -21155.749,E2 -21155.749} C_VEL
LIN {X 0,Y 212.541,Z 401.679,A -85,B 0,C 180,E1 -21158.081,E2 -21158.081} C_VEL
LIN {X 0,Y 214.56,Z 390.703,A -85,B 0,C 180,E1 -21160.129,E2 -21160.129} C_VEL
LIN {X 0,Y 216.254,Z 379.862,A -85,B 0,C 180,E1 -21161.721,E2 -21161.721} C_VEL
LIN {X 0,Y 217.59,Z 368.12,A -85,B 0,C 180,E1 -21163.069,E2 -21163.069} C_VEL
LIN {X 0,Y 218.899,Z 355.103,A -85,B 0,C 180,E1 -21164.113,E2 -21164.113} C_VEL
LIN {X 0,Y 219.756,Z 341.283,A -85,B 0,C 180,E1 -21164.826,E2 -21164.826} C_VEL
LIN {X 0,Y 222.129,Z 277.581,A -85,B 0,C 180,E1 -21166.809,E2 -21166.809} C_VEL
LIN {X 0,Y 214.573,Z 259.719,A -85,B 0,C 180,E1 -21168.445,E2 -21168.445} C_VEL
LIN {X 0,Y 207.744,Z 246.515,A -85,B 0,C 180,E1 -21169.93,E2 -21169.93} C_VEL
LIN {X 0,Y 206.768,Z 243.728,A -85,B 0,C 180,E1 -21170.213,E2 -21170.213} C_VEL
LIN {X 0,Y 206.734,Z 243.733,A -85,B 0,C 180,E1 -21174.078,E2 -21174.078} C_VEL
LIN {X 0,Y 206.692,Z 243.739,A -85,B 0,C 180,E1 -21178.429,E2 -21178.429} C_VEL
LIN {X 0,Y 206.7,Z 243.737,A -85,B 0,C 180,E1 -21182.96,E2 -21182.96} C_VEL
LIN {X 0,Y 206.674,Z 243.737,A -85,B 0,C 180,E1 -21187.744,E2 -21187.744} C_VEL
LIN {X 0,Y 206.637,Z 243.736,A -85,B 0,C 180,E1 -21191.56,E2 -21191.56} C_VEL
LIN {X 0,Y 206.636,Z 243.743,A -85,B 0,C 180,E1 -21195.584,E2 -21195.584} C_VEL
LIN {X 0,Y 206.652,Z 243.731,A -85,B 0,C 180,E1 -21199.746,E2 -21199.746} C_VEL
LIN {X 0,Y 206.707,Z 243.731,A -85,B 0,C 180,E1 -21204.689,E2 -21204.689} C_VEL
LIN {X 0,Y 206.704,Z 243.725,A -85,B 0,C 180,E1 -21209.335,E2 -21209.335} C_VEL
LIN {X 0,Y 206.781,Z 243.701,A -85,B 0,C 180,E1 -21212.378,E2 -21212.378} C_VEL
LIN {X 0,Y 213.912,Z 271.553,A -85,B 0,C 180,E1 -21214.303,E2 -21214.303} C_VEL
LIN {X 0,Y 210.403,Z 347.174,A -85,B 0,C 180,E1 -21218.773,E2 -21218.773} C_VEL
LIN {X 0,Y 209.682,Z 361.288,A -85,B 0,C 180,E1 -21219.998,E2 -21219.998} C_VEL
LIN {X 0,Y 208.73,Z 374.779,A -85,B 0,C 180,E1 -21221.599,E2 -21221.599} C_VEL
LIN {X 0,Y 207.85,Z 386.087,A -85,B 0,C 180,E1 -21223.296,E2 -21223.296} C_VEL
LIN {X 0,Y 206.972,Z 397.883,A -85,B 0,C 180,E1 -21225.497,E2 -21225.497} C_VEL
LIN {X 0,Y 206.192,Z 407.558,A -85,B 0,C 180,E1 -21227.7,E2 -21227.7} C_VEL
LIN {X 0,Y 205.56,Z 416.493,A -85,B 0,C 180,E1 -21230.157,E2 -21230.157} C_VEL
LIN {X 0,Y 205.107,Z 425.551,A -85,B 0,C 180,E1 -21233.21,E2 -21233.21} C_VEL
LIN {X 0,Y 204.804,Z 433.442,A -85,B 0,C 180,E1 -21236.557,E2 -21236.557} C_VEL
LIN {X 0,Y 204.713,Z 438.089,A -85,B 0,C 180,E1 -21239.016,E2 -21239.016} C_VEL
LIN {X 0,Y 204.872,Z 442.607,A -85,B 0,C 180,E1 -21241.965,E2 -21241.965} C_VEL
LIN {X 0,Y 205.453,Z 446.107,A -85,B 0,C 180,E1 -21244.905,E2 -21244.905} C_VEL
LIN {X 0,Y 206.36,Z 448.664,A -85,B 0,C 180,E1 -21247.829,E2 -21247.829} C_VEL
LIN {X 0,Y 208.107,Z 450.727,A -85,B 0,C 180,E1 -21251.69,E2 -21251.69} C_VEL
LIN {X 0,Y 210.436,Z 451.273,A -85,B 0,C 180,E1 -21254.407,E2 -21254.407} C_VEL
LIN {X 0,Y 213.319,Z 451.003,A -85,B 0,C 180,E1 -21257.248,E2 -21257.248} C_VEL
LIN {X 0,Y 217.471,Z 449.487,A -85,B 0,C 180,E1 -21260.492,E2 -21260.492} C_VEL
LIN {X 0,Y 218.971,Z 448.658,A -85,B 0,C 180,E1 -21261.98,E2 -21261.98} C_VEL
LIN {X 0,Y 220.206,Z 447.156,A -85,B 0,C 180,E1 -21264.52,E2 -21264.52} C_VEL
LIN {X 0,Y 221.908,Z 444.996,A -85,B 0,C 180,E1 -21266.973,E2 -21266.973} C_VEL
LIN {X 0,Y 224.069,Z 443.144,A -85,B 0,C 180,E1 -21268.292,E2 -21268.292} C_VEL
LIN {X 0,Y 229.203,Z 439.11,A -85,B 0,C 180,E1 -21270.393,E2 -21270.393} C_VEL
LIN {X 0,Y 236.227,Z 432.753,A -85,B 0,C 180,E1 -21272.885,E2 -21272.885} C_VEL
LIN {X 0,Y 243.891,Z 424.66,A -85,B 0,C 180,E1 -21275.192,E2 -21275.192} C_VEL
LIN {X 0,Y 250.773,Z 416.298,A -85,B 0,C 180,E1 -21277.052,E2 -21277.052} C_VEL
LIN {X 0,Y 258.035,Z 406.105,A -85,B 0,C 180,E1 -21278.788,E2 -21278.788} C_VEL
LIN {X 0,Y 265.071,Z 394.677,A -85,B 0,C 180,E1 -21280.261,E2 -21280.261} C_VEL
LIN {X 0,Y 271.646,Z 381.892,A -85,B 0,C 180,E1 -21281.526,E2 -21281.526} C_VEL
LIN {X 0,Y 276.515,Z 370.522,A -85,B 0,C 180,E1 -21282.377,E2 -21282.377} C_VEL
LIN {X 0,Y 281.514,Z 355.88,A -85,B 0,C 180,E1 -21283.2,E2 -21283.2} C_VEL
LIN {X 0,Y 283.117,Z 350.113,A -85,B 0,C 180,E1 -21283.48,E2 -21283.48} C_VEL
LIN {X 0,Y 282.983,Z 350.723,A -85,B 0,C 180,E1 -21284.665,E2 -21284.665} C_VEL
LIN {X 0,Y 282.924,Z 351.06,A -85,B 0,C 180,E1 -21284.87,E2 -21284.87} C_VEL
LIN {X 0,Y 278.088,Z 366.95,A -85,B 0,C 180,E1 -21285.594,E2 -21285.594} C_VEL
LIN {X 0,Y 272.437,Z 381.122,A -85,B 0,C 180,E1 -21286.362,E2 -21286.362} C_VEL
LIN {X 0,Y 265.89,Z 394.586,A -85,B 0,C 180,E1 -21287.363,E2 -21287.363} C_VEL
LIN {X 0,Y 258.868,Z 406.77,A -85,B 0,C 180,E1 -21288.564,E2 -21288.564} C_VEL
LIN {X 0,Y 251.593,Z 417.698,A -85,B 0,C 180,E1 -21290.021,E2 -21290.021} C_VEL
LIN {X 0,Y 245.315,Z 426.091,A -85,B 0,C 180,E1 -21291.454,E2 -21291.454} C_VEL
LIN {X 0,Y 238.183,Z 434.633,A -85,B 0,C 180,E1 -21293.306,E2 -21293.306} C_VEL
LIN {X 0,Y 231.073,Z 442.317,A -85,B 0,C 180,E1 -21295.493,E2 -21295.493} C_VEL
LIN {X 0,Y 224.533,Z 448.651,A -85,B 0,C 180,E1 -21297.85,E2 -21297.85} C_VEL
LIN {X 0,Y 219.058,Z 453.416,A -85,B 0,C 180,E1 -21300.177,E2 -21300.177} C_VEL
LIN {X 0,Y 212.584,Z 458.374,A -85,B 0,C 180,E1 -21303.491,E2 -21303.491} C_VEL
LIN {X 0,Y 208.531,Z 461.088,A -85,B 0,C 180,E1 -21306.142,E2 -21306.142} C_VEL
LIN {X 0,Y 204.146,Z 463.462,A -85,B 0,C 180,E1 -21309.861,E2 -21309.861} C_VEL
LIN {X 0,Y 200.763,Z 464.432,A -85,B 0,C 180,E1 -21313.734,E2 -21313.734} C_VEL
LIN {X 0,Y 198.782,Z 464.039,A -85,B 0,C 180,E1 -21317.75,E2 -21317.75} C_VEL
LIN {X 0,Y 197.944,Z 462.257,A -85,B 0,C 180,E1 -21321.833,E2 -21321.833} C_VEL
